(* CODESYS project CoreComponents.library
   Version: 1.3.1
   Title: CoreComponents
   DefaultNamespace: CoreComponents
   Placeholder: CoreComponents
   Company: Beckhoff Automation LLC

Project tree, tasks and I/O mapping:
  libraries: Tc2_DataExchange, * (Beckhoff Automation GmbH); Tc2_EtherCAT, * (Beckhoff Automation GmbH); Tc2_IoFunctions, * (Beckhoff Automation GmbH); Tc2_Math, * (Beckhoff Automation GmbH); Tc2_SerialCom, * (Beckhoff Automation GmbH); Tc2_Standard, * (Beckhoff Automation GmbH); Tc2_System, * (Beckhoff Automation GmbH); Tc2_TcpIp, * (Beckhoff Automation GmbH); Tc2_Utilities, * (Beckhoff Automation GmbH); Tc3_EventLogger, * (Beckhoff Automation GmbH); Tc3_JsonXml, * (Beckhoff Automation GmbH); Tc3_Module, * (Beckhoff Automation GmbH); Core, 1.3.0 (Beckhoff Automation LLC)
  Components/
    ADS/
      Interface/
        interface I_AdsAccess: AdsRW
        interface I_AdsRW: AmsNetId, AmsPort, Read, ReadBySymbol, Write, WriteBySymbol
      function block AdsReadWrite [ST]: Busy, Error, ErrorId, AdsComMode, AmsNetId, AmsPort, CyclicLogic, Read, ReadBySymbol, Write, WriteBySymbol
    Analog/
      DUT/
        data type ST_AnalogInputStatus_EL30xx
        data type ST_AnalogInputStatus_Generic
      Interface/
        interface I_AnalogChannel_Generic: DataValid, Error, Overrange, Underrange
        interface I_AnalogChannel_Standard: Limit1High, Limit1Low, Limit2High, Limit2Low
        interface I_AnalogInput: RawValue, Value
        interface I_AnalogOutput: RawValue, Value
      function block AnalogInput [ST]: CalibrateCustom, CalibrateLinear, FB_Init, Force, ForceValue, RawValue, Scale, Value
      function block AnalogInput_Generic [ST]: DataValid, Error, FB_Init, Overrange, Underrange
      function block AnalogInput_Standard [ST]: DataValid, Error, FB_Init, Limit1High, Limit1Low, Limit2High, Limit2Low, Overrange, Underrange
      function block AnalogOutput [ST]: CalibrateCustom, CalibrateLinear, FB_Init, Force, ForceValue, RawValue, Scale, Value
    CoE/
      DUT/
        data type ST_TerminalProductInfo
      Interface/
        interface I_CoeAccess: CoE
        interface I_CoeDevice: AdsAddr, Read, Write
      function block CoeDevice [ST]: Busy, Error, ErrorId, AdsAddr, CyclicLogic, Read, Write
      function block NullCoeDevice [ST]: AdsAddr, Busy, CyclicLogic, Error, ErrorId, Read, Write
    Cylinder/
      DUT/
        data type E_CylinderErrorId
        data type E_CylinderState
        data type ST_Cylinder_HMI
      Interface/
        interface I_Cylinder: ExtendTimeout, RetractTimeout
        interface I_CylinderCommand: Extend, Retract
        interface I_CylinderStatus: Extended, Extending, Retracted, Retracting
      function block Cylinder [ST]: CyclicLogic, Busy, Error, ErrorId, Extend, Extended, Extending, ExtendTimeout, Retract, Retracted, Retracting, RetractTimeout, Reset, FB_Init
      function block Cylinder_HMI [ST]: ExtendPermissive, RetractPermissive, ControlObject, CyclicLogic, ExtendCommandName, ExtendedName, FB_Init, RetractCommandName, RetractedName
      function block Cylinder_TcEvents [ST]: GetHighestActiveEventReaction, GetHighestActiveEventSeverity, Reset, SetEventReactions, CyclicLogic, FB_Init
    Digital/
      DUT/
        data type ST_DigitalInput_HMI
        data type ST_DigitalOutput_HMI
      Interface/
        interface I_DigitalInput: IsActive
        interface I_DigitalOutput: On
      Visitor/
        function block ForceVisitor [ST]: Force, VisitComponent
        function block ReleaseAllForceVisitor [ST]: ReleaseForces, VisitComponent, VisitModule
      function block DigitalInput_Combiner [ST]: AddInput, Force, IsActive
      function block DigitalInput_DebounceFallingEdge [ST]: CyclicLogic, DebounceTime, FB_Init, Force, IsActive
      function block DigitalInput_DebounceRisingEdge [ST]: CyclicLogic, DebounceTime, FB_Init, Force, IsActive
      function block DigitalInput_HMI [ST]: ControlObject, CyclicLogic, FB_Init
      function block DigitalInput_NC [ST]: FB_Init, Force, IsActive
      function block DigitalInput_NO [ST]: FB_Init, Force, IsActive
      function block DigitalOutput [ST]: FB_Init, Force, On
      function block DigitalOutput_HMI [ST]: ControlObject, CyclicLogic, FB_Init
    EtherCat/
      DUT/
        global variables EtherCatParameter
        data type ST_EtherCatMasterInfo
        data type ST_EtherCatSyncUnitTaskInfo
      Interface/
        interface I_EcIoDevice: Bootstrap, Configuration, DeviceError, Disabled, Init, InitCmdError, InvalidVPRS, OP, PreOp, SafeOp, State
        interface I_EtherCatDiagnosticEventProvider: RaiseEtherCatDiagnosticEvent, RaiseSyncUnitEvent
        interface I_EtherCatMasterDiagnostic: ConfiguredSlaveCount, GetIoDeviceByAddr, GetIoDeviceByName, LocalAmsNetId, MasterAmsNetId, RegisterEventProvider, SlaveCount
        interface I_IoDevice: IoDataValid
        interface I_SyncUnitTask: IoDataValid, IsHotConnect, SlaveCount
      function block EtherCatIoDevice [ST]: Bootstrap, CoE, Configuration, DeviceError, Disabled, Init, InitCmdError, InvalidVPRS, IoDataValid, OP, PreOp, SafeOp, State, AmsNetId, CyclicLogic, SyncUnit
      function block EtherCatMaster [ST]: FramesWcStatesOk, LookupMasterState, LookupSlaveState, MasterState, SlaveState, ConfiguredSlaveCount, GetIoDeviceByAddr, GetIoDeviceByName, LocalAmsNetId, MasterAmsNetId, RegisterEventProvider, SlaveCount, Initialize, Initialized, Reset, Busy, Error, ErrorId, CyclicLogic, FB_Init, Simulated
      function block EtherCatMaster_TcEvents [ST]: GetHighestActiveEventReaction, GetHighestActiveEventSeverity, RaiseEtherCatDiagnosticEvent, RaiseSyncUnitEvent, Reset, SetEventReactions, FB_Init
      function block SyncUnitTask [ST]: Initialize, Initialized, IoDataValid, IsHotConnect, IsTerminalPartOfSyncUnit, SlaveCount, Busy, Error, ErrorId, CyclicLogic, EventProvider, FB_Init, Simulated
    Recipe/
      Interface/
        interface I_RecipeManagment: AutoLoadChangesToActive, ChangesPending, LoadChangesToActive
      function block RecipeManagment [ST]: CyclicLogic, CompareData, AutoLoadChangesToActive, ChangesPending, LoadChangesToActive, FB_Init
    Safety/
      DUT/
        data type E_SafetyConnection_State
        data type E_SafetyEdm_State
        data type E_SafetyEStop_State
        data type E_SafetyGroup_Diag
        data type E_SafetyGroup_State
        data type E_SafetyMon_State
        data type E_SafetyOrAnd_State
        data type ST_SafetyAddressInfo
        data type ST_SafetyDeviceInfo
        data type ST_SafetyStateDiag
      Interface/
        interface I_InSafetyGroup: SafetyGroup
        interface I_SafetyBase: OK, ResetFunction
        interface I_SafetyModule: AddSafetyComponent, OK, SafetyPlcCoE
        interface I_SafetyReset: Execute, PulseDuration
        interface I_SafetySimulation: SimulateSafetyDiag, SimulateSafetyState
      Reset Function/
        function block SafetyResetPulse [ST]: CyclicLogic, Busy, Error, ErrorId, Execute, PulseDuration
      Visitor/
        function block SafetyOkVisitor [ST]: Check, OK, VisitComponent
        function block SetSafetySimulationVisitor [ST]: Diag, Simulated, State, VisitComponent
      function block SafetyAndOrFB [ST]: CyclicLogic
      function block SafetyBase [ST]: CyclicLogic, OK, Reset, ResetFunction, Simulated, SimulateSafetyDiag, SimulateSafetyState, Busy, Error, ErrorId
      function block SafetyConnectionFB_TcEvents [ST]: CyclicLogic, GetHighestActiveEventReaction, GetHighestActiveEventSeverity, Reset, SetEventReactions, FB_Init
      function block SafetyEdmFB_TcEvents [ST]: CyclicLogic, GetHighestActiveEventReaction, GetHighestActiveEventSeverity, Reset, SetEventReactions, FB_Init, SafetyGroup
      function block SafetyEstopFB_TcEvents [ST]: CyclicLogic, GetHighestActiveEventReaction, GetHighestActiveEventSeverity, Reset, SetEventReactions, ActiveName, FB_Init, SafetyGroup
      function block SafetyGroup_TcEvents [ST]: CyclicLogic, GetHighestActiveEventReaction, GetHighestActiveEventSeverity, Reset, SetEventReactions, AutoResetFaults, FB_Init
      function block SafetyModule [ST]: OnCyclicCall, Initializing, Simulated, SimulateSafetyDiag, SimulateSafetyState, Busy, Error, ErrorId, AddSafetyComponent, FB_Init, OK, Reset, SafetyAddressInfo, SafetyPlcCoE
      function block SafetyMonFB_TcEvents [ST]: CyclicLogic, GetHighestActiveEventReaction, GetHighestActiveEventSeverity, Reset, SetEventReactions, ActiveAlarm, ActiveName, FB_Init, SafetyGroup
    Serial/
      Interface/
        interface I_SerialByteConnection: ByteData, ByteDataRecieved, SendAByte
        interface I_SerialLineControl: rxBuffer, txBuffer
        interface I_SerialStringConnection: SendAString, StringData, StringRecieved
      function block SerialByteConnection [ST]: ByteData, ByteDataRecieved, CyclicLogic, FB_Init, Reset, SendAByte, SetDependencies
      function block SerialLineControl_ADS [ST]: CyclicLogic, rxBuffer, SetConnectionConfig, txBuffer
      function block SerialLineControl_Terminal [ST]: CyclicLogic, FB_Init, rxBuffer, SetConnectionConfig, SetDependencies, txBuffer
      function block SerialStringConnection [ST]: CyclicLogic, FB_Init, Reset, SendAString, SetDependencies, SetSerialConfiguration, StringData, StringRecieved
    Tcp Ip/
      DUT/
        data type ST_TcpIpPayload
      Interface/
        interface I_TcpIpConnection: ConnectionState, IP, Port, RegisterCommand, SendCommand, SendPriorityCommand, Socket
        interface I_TcpIpSubscription: UpdateCommandResult
      function block TcpIpCommandResultFilter [ST]: CyclicLogic, FB_Init, UpdateCommandResult
      function block TcpIpConnection [ST]: CyclicLogic, Initialize, Initialized, EvaluateResponse, GetNextCommand, GetNextPriorityCommand, SendReceiveSequence, ConnectionState, IP, PollTime, Port, ReceiveTimeout, ReconnectionTime, RegisterCommand, SendCommand, SendInterval, SendPriorityCommand, Socket
      global variables TcpIpConnectionParameter
  Project Information/
    function F_GetCompany [ST]
    function F_GetTitle [ST]
    function F_GetVersion [ST]
  Utilities/
    AnyBuffer/
      DUT/
        data type ST_BufferConfiguration
        data type ST_BufferMetadata
      Interface/
        interface I_AnyBuffer: Clear, Configuration, DeleteAtIndex, isEmpty, isFull, Metadata, PeekAtIndex, PopAtIndex, PopLeft, PopRight, PushAtIndex, PushLeft, PushRight, ReplaceAtIndex
        interface I_AnyBufferStrategy: Clear, isEmpty, isFull
      TypedBuffers/
        function block FifoBuffer [ST]: Clear, FB_Init, isEmpty, isFull, Pop, Push
        function block LifoBuffer [ST]: Clear, FB_Init, isEmpty, isFull, Pop, Push
        function block ListBuffer [ST]: Clear, FB_Init, isEmpty, isFull, Pop, Push, removeOldest
        function block RingBuffer [ST]: AdvanceHead, AdvanceTail, Clear, FB_Init, isEmpty, isFull, Pop, Push
      function block AnyBuffer [ST]: buffer, Clear, Configuration, CountDecrement, CountIncrement, DeleteAtIndex, FB_Exit, FB_Init, FB_Reinit, isEmpty, isFull, Metadata, PeekAtIndex, PopAtIndex, PopLeft, PopRight, PushAtIndex, PushLeft, PushRight, ReplaceAtIndex
    File/
      DUT/
        data type ST_File_HMI
      Interface/
        interface I_FileHandler: ClearDocument, Datatype, LoadFile, nData, Path, pData, ReadSymbol, SaveFile, SymbolName, Timeout, UpdateSymbol
      function block File_HMI [ST]: LoadPermissive, SavePermissive, ControlObject, CyclicLogic, FB_Init
      function block JsonFile [ST]: CyclicLogic, ClearDocument, Datatype, LoadFile, nData, Path, pData, ReadSymbol, SaveFile, SymbolName, Timeout, UpdateSymbol, LoadFileSequence, SaveFileSequence, Reset, Busy, Error, ErrorId
      function block StringHelper [ST]: GetExtensionOrVarName, GetFileNameFromPath, GetFilePath, GetName, GetPath, GetSymbolPath, RemoveFirstChar, RemoveLastChar, StringToCharArray, ValidInput
    Flash/
      function block SyncedSquareWaves [ST]: Initialize, Initialized, CyclicLogic, Wave_0_5Hz, Wave_100Hz, Wave_1Hz, Wave_2Hz, Wave_500Hz, Wave_50Hz, Wave_5Hz
    Force/
      DUT/
        data type E_ForceState
      Interface/
        interface I_ForcibleBool: Force
        interface I_ForcibleInt: Force, ForceValue
      function block ForcibleBool [ST]: ResolveOutput, CurrentForceState, FB_Init, Input, Output, SetForceState
      function block ForcibleInt [ST]: ResolveOutput, CurrentForceState, FB_Init, ForceValue, Input, Output, SetForceState
    Functions/
      function CompareLREAL [ST]
      function CompareModulo [ST]
      function PercentToAnalog [ST]
    Scaling/
      Interface/
        interface I_AnalogScalable: Scale
        interface I_AnalogScale: InputMaximum, InputMinimum, OutputMaximum, OutputMinimum
        interface I_CalibratableLinear: CalibrateLinear
        interface I_CalibrateLinear: Gain, Offset
        interface I_TransformLRealValue: Transform
      function block AnalogScale [ST]: InputMaximum, InputMinimum, OutputMaximum, OutputMinimum, Transform
      function block Calibrate [ST]: Gain, Offset, Transform
    Timing/
      function block Stopwatch [ST]: Elapsed, Lap, Running, Start, Stop
  Version/
    global variables Global_Version
*)

// Components/Analog/DUT/ST_AnalogInputStatus_EL30xx
{attribute 'pack_mode' := '1'}
TYPE ST_AnalogInputStatus_EL30xx :
	STRUCT
		Underrrange : BIT;
		Overrange	: BIT;
		Limit1L		: BIT;
		Limit1H		: BIT;
		Limit2L		: BIT;
		Limit2H		: BIT;
		Error		: BIT;
		TxPDOState	: BIT;
		TxPDOToggle : BIT;
	END_STRUCT
END_TYPE

// Components/Analog/DUT/ST_AnalogInputStatus_Generic
{attribute 'pack_mode' := '1'}
TYPE ST_AnalogInputStatus_Generic :
	STRUCT
		Underrrange : BIT;
		Overrange	: BIT;
		Error		: BIT;
		WcState		: BIT;
	END_STRUCT
END_TYPE

// Components/CoE/DUT/ST_TerminalProductInfo
{attribute 'pack_mode' := '2'}
TYPE ST_TerminalProductInfo : // Parameter 16#1018:0
	STRUCT
		Identity	 : WORD;
		VendorId	 : DINT;
		ProductCode	 : DINT;
		Revision	 : DINT;
		SerialNumber : DINT;
	END_STRUCT
END_TYPE

// Components/Cylinder/DUT/E_CylinderErrorId
{attribute 'qualified_only'}
TYPE E_CylinderErrorId : (
		NoError				  := 0,
		ExtendTimeout		  := 1,
		RetractTimeout		  := 2,
		ExtendedPlausibility  := 3,
		RetractedPlausibility := 4,
		BothSensorsActive	  := 5
	) UDINT;
END_TYPE

// Components/Cylinder/DUT/E_CylinderState
{attribute 'qualified_only'}
TYPE E_CylinderState : (
		Undefined  := 0,
		Extending  := 1,
		Extended   := 2,
		Retracting := 3,
		Retracted  := 4
	);
END_TYPE

// Components/Cylinder/DUT/ST_Cylinder_HMI
TYPE ST_Cylinder_HMI EXTENDS ST_HmiFunction :
	STRUCT
		Busy		  : BOOL;
		Error		  : BOOL;
		ErrorId		  : UDINT;
		Extended	  : BOOL;
		ExtendedName  : STRING := 'Extended';
		Retracted	  : BOOL;
		RetractedName : STRING := 'Retracted';
		Extend		  : Button;
		Retract		  : Button;
	END_STRUCT
END_TYPE

// Components/Digital/DUT/ST_DigitalInput_HMI
TYPE ST_DigitalInput_HMI EXTENDS ST_HmiFunction :
	STRUCT
		Active : BOOL;
		Force  : E_ForceState;
	END_STRUCT
END_TYPE

// Components/Digital/DUT/ST_DigitalOutput_HMI
TYPE ST_DigitalOutput_HMI EXTENDS ST_HmiFunction :
	STRUCT
		On	  : BOOL;
		Force : E_ForceState;
	END_STRUCT
END_TYPE

// Components/EtherCat/DUT/ST_EtherCatMasterInfo
TYPE ST_EtherCatMasterInfo :
	STRUCT
		AmsNetID	  : AMSNETID;
		DevID		  : UINT;
		DevState	  : UINT;
		ChangeCount	  : UINT;
		SlaveCount	  : UINT;
		CfgSlaveCount : UINT;
	END_STRUCT
END_TYPE

// Components/EtherCat/DUT/ST_EtherCatSyncUnitTaskInfo
TYPE ST_EtherCatSyncUnitTaskInfo :
	STRUCT
		WcState	   : BIT;
		ObjectId   : OTCID;
		State	   : UINT;
		SlaveCount : UINT;
	END_STRUCT
END_TYPE

// Components/Safety/DUT/E_SafetyConnection_State
{attribute 'qualified_only'}
{attribute 'strict'}
TYPE E_SafetyConnection_State : (
		Reset	   := 100,
		Session	   := 101,
		Connection := 102,
		Parameter  := 103,
		Data	   := 104,
		Shutdown   := 105,
		Deactive   := 106
	) USINT;
END_TYPE

// Components/Safety/DUT/E_SafetyEdm_State
{attribute 'qualified_only'}
TYPE E_SafetyEdm_State : (
		Invalid := 0,
		Stop	:= 2,
		Error	:= 4,
		Reset	:= 5,
		MonOff	:= 14,
		MonOn	:= 15
	) USINT;
END_TYPE

// Components/Safety/DUT/E_SafetyEStop_State
{attribute 'qualified_only'}
TYPE E_SafetyEStop_State : (
		Invalid	 := 0,
		Run		 := 1,
		Stop	 := 2,
		Safe	 := 3,
		Error	 := 4,
		Reset	 := 5,
		Start	 := 6,
		DelayOut := 7
	) USINT;
END_TYPE

// Components/Safety/DUT/E_SafetyGroup_Diag
{attribute 'qualified_only'}
TYPE E_SafetyGroup_Diag : (
		NoError		  := 0,
		FbError		  := 1,
		ComError	  := 2,
		ModuleError	  := 3,
		CmpError	  := 4,
		DeactiveError := 5,
		RestartError  := 6
	) UINT;
END_TYPE

// Components/Safety/DUT/E_SafetyGroup_State
{attribute 'qualified_only'}
TYPE E_SafetyGroup_State : (
		Invalid		 := 0,
		Run			 := 1,
		Stop		 := 2,
		Error		 := 4,
		Reset		 := 5,
		Start		 := 6,
		StopError	 := 7,
		Deactive	 := 16,
		WaitComError := 17
	) USINT;
END_TYPE

// Components/Safety/DUT/E_SafetyMon_State
{attribute 'qualified_only'}
TYPE E_SafetyMon_State : (
		Invalid	   := 0,
		Run		   := 1,
		Stop	   := 2,
		Safe	   := 3,
		Error	   := 4,
		Reset	   := 5,
		Start	   := 6,
		ErrorDelay := 7,
		DelayOut   := 8,
		FuncTest   := 9
	) USINT;
END_TYPE

// Components/Safety/DUT/E_SafetyOrAnd_State
{attribute 'qualified_only'}
TYPE E_SafetyOrAnd_State : (
		Invalid := 0,
		Run		:= 1,
		Stop	:= 2,
		Safe	:= 3
	) USINT;
END_TYPE

// Components/Safety/DUT/ST_SafetyAddressInfo
{attribute 'pack_mode' := '2'}
TYPE ST_SafetyAddressInfo : // Parameter 16#F980:0
	STRUCT
		FSoEAddress		  : WORD;
		SerialNumber	  : DINT;
		ProjectCRC		  : WORD;
		DefaultProjectCRC : WORD;
	END_STRUCT
END_TYPE

// Components/Safety/DUT/ST_SafetyDeviceInfo
{attribute 'pack_mode' := '2'}
TYPE ST_SafetyDeviceInfo : // Parameter 16#F9C0:0
	STRUCT
		DeviceName			 : STRING;
		SoftwareVersion		 : STRING;
		BootloaderVersion	 : STRING;
		SoftwareChecksum	 : DINT;
		BootmanagerChecksum	 : DINT;
		BootloaderChecksum	 : DINT;
		TwinSAFELogicVersion : DINT;
	END_STRUCT
END_TYPE

// Components/Safety/DUT/ST_SafetyStateDiag
{attribute 'pack_mode' := '1'}
TYPE ST_SafetyStateDiag :
	STRUCT
		State : USINT;
		Diag  : UINT; // **NOT PRESENT ON AND/OR FBs ** For components with USINT as Diag connection, connect first 8 Bit of UINT Diag. Inherited FB is evaluating correct length.
	END_STRUCT
END_TYPE

// Components/Tcp Ip/DUT/ST_TcpIpPayload
TYPE ST_TcpIpPayload :
	STRUCT
		Size : UDINT;
		Data : ARRAY[0..(TcpIpConnectionParameter.PayloadSize - 1)] OF BYTE;
	END_STRUCT
END_TYPE

// Utilities/AnyBuffer/DUT/ST_BufferConfiguration
TYPE ST_BufferConfiguration :
	STRUCT
		isPersistent	 : BOOL; // is the buffer persistent?
		capacity		 : DINT; // No of elements in buffer
		elementSize		 : DINT; // Buffer element size in bytes
		bufferSize		 : DINT; // Complete buffer size in bytes	
		bufferBoundLower : DINT; // Lower boundary of the buffer
		bufferBoundUpper : DINT; // Upper boundary of the buffer	
	END_STRUCT
END_TYPE

// Utilities/AnyBuffer/DUT/ST_BufferMetadata
TYPE ST_BufferMetadata :
	STRUCT
		headIndex	 : DINT;
		tailIndex	 : DINT;
		capacity	 : DINT;
		elementCount : DINT;
	END_STRUCT
END_TYPE

// Utilities/File/DUT/ST_File_HMI
TYPE ST_File_HMI EXTENDS ST_HmiFunction :
	STRUCT
		Path	: STRING;
		Load	: Button;
		Save	: Button;
		NewPath : BOOL;
	END_STRUCT
END_TYPE

// Utilities/Force/DUT/E_ForceState
{attribute 'qualified_only'}
{attribute 'strict'}
{attribute 'to_string'}
TYPE E_ForceState : (
		Unforced := 0,
		ForceOn	 := 1,
		ForceOff := 2
	) DINT;
END_TYPE

// Components/EtherCat/DUT/EtherCatParameter
VAR_GLOBAL CONSTANT
	MAX_EC_SLAVES : UINT := 49;
END_VAR

// Components/Tcp Ip/TcpIpConnectionParameter
{attribute 'qualified_only'}
VAR_GLOBAL CONSTANT
	PayloadSize : UDINT := 1460; // Payload in Bytes
END_VAR

// Version/Global_Version
{attribute 'TcGenerated'}
{attribute 'no-analysis'}
{attribute 'linkalways'}
// This function has been automatically generated from the project information.
VAR_GLOBAL CONSTANT
	{attribute 'const_non_replaced'}
	stLibVersion_CoreComponents : ST_LibVersion := (iMajor := 1, iMinor := 3, iBuild := 1, iRevision := 0, nFlags := 0, sVersion := '1.3.1');
END_VAR

// Components/ADS/Interface/I_AdsAccess
INTERFACE I_AdsAccess EXTENDS I_Base

PROPERTY AdsRW : I_AdsRW
GET
END_GET
SET
END_SET
END_PROPERTY

END_INTERFACE

// Components/ADS/Interface/I_AdsRW
INTERFACE I_AdsRW EXTENDS I_Component, I_TaskResult

{attribute 'monitoring' := 'call'}
PROPERTY AmsNetId : T_AmsNetId
GET
END_GET
SET
END_SET
END_PROPERTY

{attribute 'monitoring' := 'call'}
PROPERTY AmsPort : T_AmsPort
GET
END_GET
SET
END_SET
END_PROPERTY

METHOD Read
VAR_INPUT
	IdxGrp	  : UDINT;
	IdxOffset : UDINT;
	pDestAddr : PVOID;
	Length	  : UDINT;
END_VAR
END_METHOD

METHOD ReadBySymbol
VAR_INPUT
	SymbolName : STRING(255);
	pDestAddr  : PVOID;
	Length	   : UDINT;
END_VAR
END_METHOD

METHOD Write
VAR_INPUT
	IdxGrp		: UDINT;
	IdxOffset	: UDINT;
	pSourceAddr : PVOID;
	Length		: UDINT;
END_VAR
END_METHOD

METHOD WriteBySymbol
VAR_INPUT
	SymbolName	: STRING(255);
	pSourceAddr : PVOID;
	Length		: UDINT;
END_VAR
END_METHOD

END_INTERFACE

// Components/ADS/AdsReadWrite
FUNCTION_BLOCK AdsReadWrite EXTENDS CyclicComponent IMPLEMENTS I_AdsRW
VAR
	{attribute 'hide'}
	_AmsNetId : T_AmsNetId;
	{attribute 'hide'}
	_AmsPort : T_AmsPort;
	{attribute 'hide'}
	_AdsComMode		  : E_AdsComMode := eAdsComModeSecureCom;
	AdsRead			  : ADSREAD;
	AdsWrite		  : ADSWRITE;
	ReadAdsSymByName  : FB_ReadAdsSymByName;
	WriteAdsSymByName : FB_WriteAdsSymByName;
END_VAR

{attribute 'monitoring' := 'call'}
PROPERTY Busy : BOOL
GET
Busy := AdsWrite.BUSY OR AdsRead.BUSY OR ReadAdsSymByName.bBusy OR WriteAdsSymByName.bBusy;
END_GET
END_PROPERTY

{attribute 'monitoring' := 'call'}
PROPERTY Error : BOOL
GET
Error := AdsWrite.ERR OR AdsRead.ERR OR ReadAdsSymByName.bError OR WriteAdsSymByName.bError;
END_GET
END_PROPERTY

{attribute 'monitoring' := 'call'}
PROPERTY ErrorId : UDINT
GET
IF AdsWrite.ERR THEN
	ErrorID := AdsWrite.ERRID;
ELSIF AdsRead.ERR THEN
	ErrorID := AdsRead.ERRID;
ELSIF ReadAdsSymByName.bError THEN
	ErrorID := ReadAdsSymByName.nErrorId;
ELSIF WriteAdsSymByName.bError THEN
	ErrorID := WriteAdsSymByName.nErrorId;
ELSE
	ErrorID := 0;
END_IF
END_GET
END_PROPERTY

PROPERTY AdsComMode : E_AdsComMode
SET
_AdsComMode := AdsComMode;
END_SET
END_PROPERTY

{attribute 'monitoring' := 'call'}
PROPERTY AmsNetId : T_AmsNetId
GET
AmsNetId := _AmsNetId;
END_GET
SET
_AmsNetId := AmsNetId;
END_SET
END_PROPERTY

{attribute 'monitoring' := 'call'}
PROPERTY AmsPort : T_AmsPort
GET
AmsPort := _AmsPort;
END_GET
SET
_AmsPort := AmsPort;
END_SET
END_PROPERTY

METHOD CyclicLogic
AdsRead(NETID := _AmsNetId, PORT := _AmsPort, TMOUT := DEFAULT_ADS_TIMEOUT);
AdsRead.READ := FALSE;
AdsWrite(NETID := _AmsNetId, PORT := _AmsPort, TMOUT := DEFAULT_ADS_TIMEOUT);
AdsWrite.WRITE := FALSE;

//
ReadAdsSymByName(sNetId		   := _AmsNetId,
				 nPort		   := _AmsPort,
				 tTimeout	   := DEFAULT_ADS_TIMEOUT,
				 eComMode	   := _AdsComMode,
				 bClearOnError := TRUE);

ReadAdsSymByName.bRead := FALSE;

//
WriteAdsSymByName(sNetId   := _AmsNetId,
				  nPort	   := _AmsPort,
				  tTimeout := DEFAULT_ADS_TIMEOUT,
				  eComMode := _AdsComMode);

WriteAdsSymByName.bWrite := FALSE;
END_METHOD

METHOD Read
VAR_INPUT
	IdxGrp	  : UDINT;
	IdxOffset : UDINT;
	pDestAddr : PVOID;
	Length	  : UDINT;
END_VAR
IF AdsRead.BUSY THEN
	RETURN;
END_IF

AdsRead.IDXGRP	 := IdxGrp;
AdsRead.IDXOFFS	 := IdxOffset;
AdsRead.LEN		 := Length;
AdsRead.DESTADDR := pDestAddr;
AdsRead.READ	 := TRUE;
END_METHOD

METHOD ReadBySymbol
VAR_INPUT
	SymbolName : STRING(255);
	pDestAddr  : PVOID;
	Length	   : UDINT;
END_VAR
IF ReadAdsSymByName.bBusy THEN
	RETURN;
END_IF

ReadAdsSymByName.sVarName  := SymbolName;
ReadAdsSymByName.nDestAddr := pDestAddr;
ReadAdsSymByName.nLen	   := Length;
ReadAdsSymByName.bRead	   := TRUE;
END_METHOD

METHOD Write
VAR_INPUT
	IdxGrp		: UDINT;
	IdxOffset	: UDINT;
	pSourceAddr : PVOID;
	Length		: UDINT;
END_VAR
IF AdsWrite.BUSY THEN
	RETURN;
END_IF

AdsWrite.IDXGRP	 := IdxGrp;
AdsWrite.IDXOFFS := IdxOffset;
AdsWrite.LEN	 := Length;
AdsWrite.SRCADDR := pSourceAddr;
AdsWrite.WRITE	 := TRUE;
END_METHOD

METHOD WriteBySymbol
VAR_INPUT
	SymbolName	: STRING(255);
	pSourceAddr : PVOID;
	Length		: UDINT;
END_VAR
IF WriteAdsSymByName.bBusy THEN
	RETURN;
END_IF

WriteAdsSymByName.sVarName := SymbolName;
WriteAdsSymByName.nSrcAddr := pSourceAddr;
WriteAdsSymByName.nLen	   := Length;
WriteAdsSymByName.bWrite   := TRUE;
END_METHOD

END_FUNCTION_BLOCK

// Components/Analog/Interface/I_AnalogChannel_Generic
INTERFACE I_AnalogChannel_Generic EXTENDS I_AnalogInput

PROPERTY DataValid : BOOL
GET
END_GET
END_PROPERTY

PROPERTY Error : BOOL
GET
END_GET
END_PROPERTY

PROPERTY Overrange : BOOL
GET
END_GET
END_PROPERTY

PROPERTY Underrange : BOOL
GET
END_GET
END_PROPERTY

END_INTERFACE

// Components/Analog/Interface/I_AnalogInput
INTERFACE I_AnalogInput EXTENDS I_Component, I_ForcibleInt

{attribute 'monitoring' := 'call'}
PROPERTY RawValue : INT
GET
END_GET
END_PROPERTY

{attribute 'monitoring' := 'call'}
PROPERTY Value : LREAL
GET
END_GET
END_PROPERTY

END_INTERFACE

// Utilities/Force/Interface/I_ForcibleInt
INTERFACE I_ForcibleInt

{attribute 'monitoring' := 'call'}
PROPERTY Force : E_ForceState
GET
END_GET
SET
END_SET
END_PROPERTY

PROPERTY ForceValue : INT
GET
END_GET
SET
END_SET
END_PROPERTY

END_INTERFACE

// Components/Analog/Interface/I_AnalogChannel_Standard
INTERFACE I_AnalogChannel_Standard EXTENDS I_AnalogChannel_Generic

PROPERTY Limit1High : BOOL
GET
END_GET
END_PROPERTY

PROPERTY Limit1Low : BOOL
GET
END_GET
END_PROPERTY

PROPERTY Limit2High : BOOL
GET
END_GET
END_PROPERTY

PROPERTY Limit2Low : BOOL
GET
END_GET
END_PROPERTY

END_INTERFACE

// Components/Analog/Interface/I_AnalogOutput
INTERFACE I_AnalogOutput EXTENDS I_Component, I_ForcibleInt

{attribute 'monitoring' := 'call'}
PROPERTY RawValue : INT
GET
END_GET
SET
END_SET
END_PROPERTY

{attribute 'monitoring' := 'call'}
PROPERTY Value : LREAL
GET
END_GET
SET
END_SET
END_PROPERTY

END_INTERFACE

// Components/Analog/AnalogInput
FUNCTION_BLOCK AnalogInput EXTENDS Component IMPLEMENTS I_AnalogInput, I_AnalogScalable, I_CalibratableLinear
VAR
	Input			 : REFERENCE TO INT;
	Forcible		 : ForcibleInt(_Name);
	_Scale			 : I_AnalogScale;
	_CalibrateLinear : I_CalibrateLinear;
	_CalibrateCustom : I_TransformLRealValue;
END_VAR

VAR
	{attribute 'hide'}
	DefaultScale : AnalogScale;
	{attribute 'hide'}
	DefaultCalibration : Calibrate;
END_VAR

PROPERTY CalibrateCustom : I_TransformLrealValue
SET
_CalibrateCustom := CalibrateCustom;
END_SET
END_PROPERTY

PROPERTY CalibrateLinear : I_CalibrateLinear
GET
CalibrateLinear := _CalibrateLinear;
END_GET
SET
_CalibrateLinear := CalibrateLinear;
END_SET
END_PROPERTY

(*FB_Init is always available implicitly and it is used primarily for initialization.
The return value is not evaluated. For a specific influence, you can also declare the
methods explicitly and provide additional code there with the standard initialization
code. You can evaluate the return value.*)
METHOD FB_Init : BOOL
VAR_INPUT
	(* TRUE: the retain variables are initialized (reset warm / reset cold)*)
	bInitRetains : BOOL;

	(* TRUE: the instance will be copied to the copy code afterward (online change)   *)
	bInCopyCode : BOOL;
	Name		: Core.T_MaxString;
	Input		: REFERENCE TO INT;
END_VAR
_Scale			 := DefaultScale;
_CalibrateLinear := DefaultCalibration;
THIS^.Input		 REF= Input;
END_METHOD

{attribute 'monitoring' := 'call'}
PROPERTY Force : E_ForceState
GET
Force := Forcible.CurrentForceState;
END_GET
SET
VAR
	ForceString : T_MaxString := TO_STRING(Force);
END_VAR
Forcible.SetForceState(Force);
END_SET
END_PROPERTY

PROPERTY ForceValue : INT
GET
ForceValue := Forcible.ForceValue;
END_GET
SET
Forcible.ForceValue := ForceValue;
END_SET
END_PROPERTY

{attribute 'monitoring' := 'call'}
PROPERTY RawValue : INT
GET
Forcible.Input := Input;
RawValue	   := Forcible.Output;
END_GET
END_PROPERTY

PROPERTY Scale : I_AnalogScale
GET
Scale := _Scale;
END_GET
SET
_Scale := Scale;
END_SET
END_PROPERTY

{attribute 'monitoring' := 'call'}
PROPERTY Value : LREAL
GET
IF _CalibrateCustom = 0 THEN
	Value := _CalibrateLinear.Transform(_Scale.Transform(RawValue));
ELSE
	Value := _CalibrateCustom.Transform(_Scale.Transform(RawValue));
END_IF
END_GET
END_PROPERTY

END_FUNCTION_BLOCK

// Utilities/Scaling/Interface/I_AnalogScalable
INTERFACE I_AnalogScalable EXTENDS I_Base

PROPERTY Scale : I_AnalogScale
GET
END_GET
SET
END_SET
END_PROPERTY

END_INTERFACE

// Utilities/Scaling/Interface/I_AnalogScale
INTERFACE I_AnalogScale EXTENDS I_TransformLrealValue

PROPERTY InputMaximum : LREAL
GET
END_GET
SET
END_SET
END_PROPERTY

PROPERTY InputMinimum : LREAL
GET
END_GET
SET
END_SET
END_PROPERTY

PROPERTY OutputMaximum : LREAL
GET
END_GET
SET
END_SET
END_PROPERTY

PROPERTY OutputMinimum : LREAL
GET
END_GET
SET
END_SET
END_PROPERTY

END_INTERFACE

// Utilities/Scaling/Interface/I_TransformLRealValue
INTERFACE I_TransformLRealValue EXTENDS I_Base

METHOD Transform : LREAL
VAR_INPUT
	Value	: LREAL;
	Reverse : BOOL := FALSE;
END_VAR
END_METHOD

END_INTERFACE

// Utilities/Scaling/Interface/I_CalibratableLinear
INTERFACE I_CalibratableLinear EXTENDS I_Base

PROPERTY CalibrateLinear : I_CalibrateLinear
GET
END_GET
SET
END_SET
END_PROPERTY

END_INTERFACE

// Utilities/Scaling/Interface/I_CalibrateLinear
INTERFACE I_CalibrateLinear EXTENDS I_TransformLrealValue

PROPERTY Gain : LREAL
SET
END_SET
END_PROPERTY

PROPERTY Offset : LREAL
SET
END_SET
END_PROPERTY

END_INTERFACE

// Utilities/Force/ForcibleInt
FUNCTION_BLOCK ForcibleInt
VAR
	Name			   : T_MaxString;
	_CurrentForceState : E_ForceState;
	ForceEvent		   : FB_TcAlarm;
	RequestedValue	   : INT;
	_Output			   : INT;
	_ForceValue : INT;
END_VAR

METHOD PRIVATE ResolveOutput
VAR
	ForceString : T_MaxString := TO_STRING(_CurrentForceState);
END_VAR
CASE _CurrentForceState OF
	E_ForceState.Unforced:
		_Output := RequestedValue;
		ForceEvent.Clear();

	E_ForceState.ForceOn:
		IF NOT ForceEvent.bActive THEN
			ForceEvent.ipArguments.Clear().AddString(Name).AddString(ForceString);
			ForceEvent.Raise();
		END_IF

		_Output := _ForceValue;

	E_ForceState.ForceOff:
		IF NOT ForceEvent.bActive THEN
			ForceEvent.ipArguments.Clear().AddString(Name).AddString(ForceString);
			ForceEvent.Raise();
		END_IF

		_Output := 0;
END_CASE
END_METHOD

{attribute 'monitoring' := 'call'}
PROPERTY CurrentForceState : E_ForceState
GET
CurrentForceState := _CurrentForceState;
END_GET
END_PROPERTY

//FB_Init is always available implicitly and it is used primarily for initialization.

//The return value is not evaluated. For a specific influence, you can also declare the

//methods explicitly and provide additional code there with the standard initialization

//code. You can evaluate the return value.
METHOD FB_Init : BOOL
VAR_INPUT
	bInitRetains : BOOL; // TRUE: the retain variables are initialized (reset warm / reset cold)
	bInCopyCode	 : BOOL; // TRUE: the instance will be copied to the copy code afterward (online change) 
	Name		 : T_MaxString;
END_VAR
THIS^.Name := Name;
{analysis -15}
IF NOT ForceEvent.EqualsToEventEntryEx(TC_EVENTS.IO.ForceActive) THEN
	ForceEvent.CreateEx(TC_EVENTS.IO.ForceActive, 0);
END_IF
END_METHOD

PROPERTY ForceValue : INT
GET
ForceValue := _ForceValue;
END_GET
SET
_ForceValue := ForceValue;
END_SET
END_PROPERTY

{attribute 'monitoring' := 'call'}
PROPERTY Input : INT
SET
RequestedValue := Input;
ResolveOutput();
END_SET
END_PROPERTY

{attribute 'monitoring' := 'call'}
PROPERTY Output : INT
GET
Output := _Output;
END_GET
END_PROPERTY

METHOD SetForceState
VAR_INPUT
	ForceState : E_ForceState;
END_VAR
IF ForceState = _CurrentForceState THEN
	RETURN;
END_IF

_CurrentForceState := ForceState;
ResolveOutput();
END_METHOD

END_FUNCTION_BLOCK

// Utilities/Scaling/AnalogScale
FUNCTION_BLOCK AnalogScale IMPLEMENTS I_AnalogScale
VAR
	_InputMinimum  : LREAL := -32768;
	_InputMaximum  : LREAL := 32767;
	_OutputMinimum : LREAL := -32768;
	_OutputMaximum : LREAL := 32767;
END_VAR

PROPERTY InputMaximum : LREAL
GET
InputMaximum := _InputMaximum;
END_GET
SET
_InputMaximum := InputMaximum;
END_SET
END_PROPERTY

PROPERTY InputMinimum : LREAL
GET
InputMinimum := _InputMinimum;
END_GET
SET
_InputMinimum := InputMinimum;
END_SET
END_PROPERTY

PROPERTY OutputMaximum : LREAL
GET
OutputMaximum := _OutputMaximum;
END_GET
SET
_OutputMaximum := OutputMaximum;
END_SET
END_PROPERTY

PROPERTY OutputMinimum : LREAL
GET
OutputMinimum := _OutputMinimum;
END_GET
SET
_OutputMinimum := OutputMinimum;
END_SET
END_PROPERTY

METHOD Transform : LREAL
VAR_INPUT
	Value	: LREAL;
	Reverse : BOOL := FALSE;
END_VAR

VAR_INST
	Slope : LREAL;
END_VAR
//Scale is invalid
IF _InputMinimum >= _InputMaximum THEN
	Transform := 0;
	RETURN;
ELSIF _OutputMinimum >= _OutputMaximum THEN
	Transform := 0;
	RETURN;
END_IF

//Input is invalid
IF Value <= _InputMinimum THEN
	Transform := _OutputMinimum;
	RETURN;
ELSIF Value >= _InputMaximum THEN
	Transform := _OutputMaximum;
	RETURN;
END_IF

//I/O ok--scale it
IF (_InputMaximum - _InputMinimum) <> 0.0 THEN
	Slope := (_OutputMaximum - _OutputMinimum) / (_InputMaximum - _InputMinimum);
ELSE
	Slope := 0.0;
END_IF

Transform := Slope * (Value - _InputMinimum) + _OutputMinimum;
END_METHOD

END_FUNCTION_BLOCK

// Utilities/Scaling/Calibrate
FUNCTION_BLOCK Calibrate IMPLEMENTS I_CalibrateLinear
VAR
	_Gain	: LREAL := 1;
	_Offset : LREAL := 0;
END_VAR

PROPERTY Gain : LREAL
SET
_Gain := Gain;
END_SET
END_PROPERTY

PROPERTY Offset : LREAL
SET
_Offset := Offset;
END_SET
END_PROPERTY

METHOD Transform : LREAL
VAR_INPUT
	Value	: LREAL;
	Reverse : BOOL := FALSE;
END_VAR
IF Reverse THEN
	Transform := (Value - _Offset) / _Gain;
ELSE
	Transform := Value * _Gain + _Offset;
END_IF
END_METHOD

END_FUNCTION_BLOCK

// Components/Analog/AnalogInput_Generic
FUNCTION_BLOCK AnalogInput_Generic EXTENDS AnalogInput IMPLEMENTS I_AnalogChannel_Generic
VAR
	Status : REFERENCE TO ST_AnalogInputStatus_Generic;
END_VAR

PROPERTY DataValid : BOOL
GET
DataValid := NOT Status.WcState;
END_GET
END_PROPERTY

PROPERTY Error : BOOL
GET
Error := Status.Error;
END_GET
END_PROPERTY

(*FB_Init is always available implicitly and it is used primarily for initialization.
The return value is not evaluated. For a specific influence, you can also declare the
methods explicitly and provide additional code there with the standard initialization
code. You can evaluate the return value.*)
METHOD FB_Init : BOOL
VAR_INPUT
	(* TRUE: the retain variables are initialized (reset warm / reset cold)*)
	bInitRetains : BOOL;

	(* TRUE: the instance will be copied to the copy code afterward (online change)   *)
	bInCopyCode : BOOL;
	Name		: T_MaxString;
	Input		: REFERENCE TO INT;
	Status		: REFERENCE TO ST_AnalogInputStatus_Generic;
END_VAR
THIS^.Status REF= Status;
END_METHOD

PROPERTY Overrange : BOOL
GET
Overrange := Status.Overrange;
END_GET
END_PROPERTY

PROPERTY Underrange : BOOL
GET
Underrange := Status.Underrrange;
END_GET
END_PROPERTY

END_FUNCTION_BLOCK

// Components/Analog/AnalogInput_Standard
FUNCTION_BLOCK AnalogInput_Standard EXTENDS AnalogInput IMPLEMENTS I_AnalogChannel_Standard
VAR
	Status : REFERENCE TO ST_AnalogInputStatus_EL30xx;
END_VAR

PROPERTY DataValid : BOOL
GET
DataValid := NOT Status.TxPDOState;
END_GET
END_PROPERTY

PROPERTY Error : BOOL
GET
Error := Status.Error;
END_GET
END_PROPERTY

(*FB_Init is always available implicitly and it is used primarily for initialization.
The return value is not evaluated. For a specific influence, you can also declare the
methods explicitly and provide additional code there with the standard initialization
code. You can evaluate the return value.*)
METHOD FB_Init : BOOL
VAR_INPUT
	(* TRUE: the retain variables are initialized (reset warm / reset cold)*)
	bInitRetains : BOOL;

	(* TRUE: the instance will be copied to the copy code afterward (online change)   *)
	bInCopyCode : BOOL;
	Name		: Core.T_MaxString;
	Input		: REFERENCE TO INT;
	Status		: REFERENCE TO ST_AnalogInputStatus_EL30xx;
END_VAR
THIS^.Status REF= Status;
END_METHOD

PROPERTY Limit1High : BOOL
GET
Limit1High := Status.Limit1H;
END_GET
END_PROPERTY

PROPERTY Limit1Low : BOOL
GET
Limit1Low := Status.Limit1L;
END_GET
END_PROPERTY

PROPERTY Limit2High : BOOL
GET
Limit2High := Status.Limit2H;
END_GET
END_PROPERTY

PROPERTY Limit2Low : BOOL
GET
Limit2Low := Status.Limit2L;
END_GET
END_PROPERTY

PROPERTY Overrange : BOOL
GET
Overrange := Status.Overrange;
END_GET
END_PROPERTY

PROPERTY Underrange : BOOL
GET
Underrange := Status.Underrrange;
END_GET
END_PROPERTY

END_FUNCTION_BLOCK

// Components/Analog/AnalogOutput
FUNCTION_BLOCK AnalogOutput EXTENDS Component IMPLEMENTS I_AnalogOutput, I_AnalogScalable, I_CalibratableLinear
VAR
	Output			 : REFERENCE TO INT;
	Forcible		 : ForcibleInt(_Name);
	_Scale			 : I_AnalogScale;
	_CalibrateLinear : I_CalibrateLinear;
	_CalibrateCustom : I_TransformLRealValue;
END_VAR

VAR
	{attribute 'hide'}
	DefaultScale : AnalogScale;
	{attribute 'hide'}
	DefaultCalibration : Calibrate;
END_VAR

PROPERTY CalibrateCustom : I_TransformLrealValue
SET
_CalibrateCustom := CalibrateCustom;
END_SET
END_PROPERTY

PROPERTY CalibrateLinear : I_CalibrateLinear
GET
CalibrateLinear := _CalibrateLinear;
END_GET
SET
_CalibrateLinear := CalibrateLinear;
END_SET
END_PROPERTY

(*FB_Init is always available implicitly and it is used primarily for initialization.
The return value is not evaluated. For a specific influence, you can also declare the
methods explicitly and provide additional code there with the standard initialization
code. You can evaluate the return value.*)
METHOD FB_Init : BOOL
VAR_INPUT
	(* TRUE: the retain variables are initialized (reset warm / reset cold)*)
	bInitRetains : BOOL;

	(* TRUE: the instance will be copied to the copy code afterward (online change)   *)
	bInCopyCode : BOOL;
	Name		: T_MaxString;
	Output		: REFERENCE TO INT;
END_VAR
_Scale			 := DefaultScale;
_CalibrateLinear := DefaultCalibration;
THIS^.Output	 REF= Output;
END_METHOD

{attribute 'monitoring' := 'call'}
PROPERTY Force : E_ForceState
GET
Force := Forcible.CurrentForceState;
END_GET
SET
VAR
	ForceString : T_MaxString := TO_STRING(Force);
END_VAR
Forcible.SetForceState(Force);
END_SET
END_PROPERTY

PROPERTY ForceValue : INT
GET
ForceValue := Forcible.ForceValue;
END_GET
SET
Forcible.ForceValue := ForceValue;
END_SET
END_PROPERTY

{attribute 'monitoring' := 'call'}
PROPERTY RawValue : INT
GET
RawValue := Output;
END_GET
SET
Forcible.Input := RawValue;
Output		   := Forcible.Output;
END_SET
END_PROPERTY

PROPERTY Scale : I_AnalogScale
GET
Scale := _Scale;
END_GET
SET
_Scale := Scale;
END_SET
END_PROPERTY

{attribute 'monitoring' := 'call'}
PROPERTY Value : LREAL
GET
IF _CalibrateCustom = 0 THEN
	Value := _CalibrateLinear.Transform(_Scale.Transform(RawValue));
ELSE
	Value := _CalibrateCustom.Transform(_Scale.Transform(RawValue));
END_IF
END_GET
SET
IF _CalibrateCustom = 0 THEN
	RawValue := LREAL_TO_INT(_Scale.Transform(_CalibrateLinear.Transform(Value, TRUE)));
ELSE
	RawValue := LREAL_TO_INT(_Scale.Transform(_CalibrateCustom.Transform(Value, TRUE)));
END_IF
END_SET
END_PROPERTY

END_FUNCTION_BLOCK

// Components/CoE/Interface/I_CoeAccess
INTERFACE I_CoeAccess EXTENDS I_Base

PROPERTY CoE : I_CoeDevice
GET
END_GET
END_PROPERTY

END_INTERFACE

// Components/CoE/Interface/I_CoeDevice
INTERFACE I_CoeDevice EXTENDS I_Component, I_TaskResult

PROPERTY AdsAddr : REFERENCE TO AMSADDR
GET
END_GET
SET
END_SET
END_PROPERTY

METHOD Read
VAR_INPUT
	Index	 : WORD;
	SubIndex : BYTE;
	pDstBuf	 : PVOID;
	BufLen	 : UDINT;
END_VAR
END_METHOD

METHOD Write
VAR_INPUT
	Index	 : WORD;
	SubIndex : BYTE;
	pDstBuf	 : PVOID;
	BufLen	 : UDINT;
END_VAR
END_METHOD

END_INTERFACE

// Components/CoE/CoeDevice
FUNCTION_BLOCK CoeDevice EXTENDS CyclicComponent IMPLEMENTS I_CoeDevice
VAR
	{attribute 'hide'}
	_Error : BOOL;
	{attribute 'hide'}
	_Busy : BOOL;
	{attribute 'hide'}
	_ErrorId : UDINT;
	_AdsAddr : REFERENCE TO AMSADDR;
	CoeRead	 : FB_EcCoESdoReadEx;
	CoeWrite : FB_EcCoESdoReadEx;
END_VAR

{attribute 'monitoring' := 'call'}
PROPERTY Busy : BOOL
GET
Busy := _Busy;
END_GET
END_PROPERTY

{attribute 'monitoring' := 'call'}
PROPERTY Error : BOOL
GET
Error := _Error;
END_GET
END_PROPERTY

{attribute 'monitoring' := 'call'}
PROPERTY ErrorId : UDINT
GET
ErrorID := _ErrorID;
END_GET
END_PROPERTY

PROPERTY AdsAddr : REFERENCE TO AMSADDR
GET
AdsAddr REF= _AdsAddr;
END_GET
SET
_AdsAddr REF= AdsAddr;
END_SET
END_PROPERTY

METHOD CyclicLogic
VAR_INST
END_VAR
IF NOT __ISVALIDREF(_AdsAddr) THEN
	RETURN;
END_IF

CoeRead(sNetId := F_CreateAmsNetId(AdsAddr.netId), nSlaveAddr := AdsAddr.port, tTimeout := T#1S);
CoeWrite(sNetId := F_CreateAmsNetId(AdsAddr.netId), nSlaveAddr := AdsAddr.port, tTimeout := T#1S);
CoeRead.bExecute  := FALSE;
CoeWrite.bExecute := FALSE;
_Busy			  := CoeRead.bBusy OR CoeWrite.bBusy;
_Error			  := CoeRead.bError OR CoeWrite.bError;
IF CoeRead.bError THEN
	_ErrorId := CoeRead.nErrId;
END_IF

IF CoeWrite.bError THEN
	_ErrorId := CoeWrite.nErrId;
END_IF
END_METHOD

METHOD Read
VAR_INPUT
	Index	 : WORD;
	SubIndex : BYTE;
	pDstBuf	 : PVOID;
	BufLen	 : UDINT;
END_VAR
IF _Busy THEN
	RETURN;
END_IF

CoeRead.nSubIndex		:= SubIndex;
CoeRead.nIndex			:= Index;
CoeRead.pDstBuf			:= pDstBuf;
CoeRead.cbBufLen		:= BufLen;
CoeRead.bCompleteAccess := SubIndex = 0;
_Busy					:= TRUE;
CoeRead.bExecute		:= TRUE;
END_METHOD

METHOD Write
VAR_INPUT
	Index	 : WORD;
	SubIndex : BYTE;
	pDstBuf	 : PVOID;
	BufLen	 : UDINT;
END_VAR
IF _Busy THEN
	RETURN;
END_IF

CoeWrite.nSubIndex		 := SubIndex;
CoeWrite.nIndex			 := Index;
CoeWrite.pDstBuf		 := pDstBuf;
CoeWrite.cbBufLen		 := BufLen;
CoeWrite.bCompleteAccess := SubIndex = 0;
_Busy					 := TRUE;
CoeWrite.bExecute		 := TRUE;
END_METHOD

END_FUNCTION_BLOCK

// Components/CoE/NullCoeDevice
FUNCTION_BLOCK NullCoeDevice EXTENDS CyclicComponent IMPLEMENTS I_CoeDevice
VAR
END_VAR

PROPERTY AdsAddr : REFERENCE TO AMSADDR
GET
END_GET
SET
END_SET
END_PROPERTY

{attribute 'monitoring' := 'call'}
PROPERTY Busy : BOOL
GET
END_GET
END_PROPERTY

METHOD CyclicLogic
END_METHOD

{attribute 'monitoring' := 'call'}
PROPERTY Error : BOOL
GET
END_GET
END_PROPERTY

{attribute 'monitoring' := 'call'}
PROPERTY ErrorId : UDINT
GET
END_GET
END_PROPERTY

METHOD Read
VAR_INPUT
	Index	 : WORD;
	SubIndex : BYTE;
	pDstBuf	 : PVOID;
	BufLen	 : UDINT;
END_VAR
END_METHOD

METHOD Write
VAR_INPUT
	Index	 : WORD;
	SubIndex : BYTE;
	pDstBuf	 : PVOID;
	BufLen	 : UDINT;
END_VAR
END_METHOD

END_FUNCTION_BLOCK

// Components/Cylinder/Interface/I_Cylinder
INTERFACE I_Cylinder EXTENDS I_CylinderCommand, I_CylinderStatus, I_Component, I_TaskResult, I_Resettable

{attribute 'monitoring' := 'call'}
PROPERTY ExtendTimeout : TIME
GET
END_GET
SET
END_SET
END_PROPERTY

{attribute 'monitoring' := 'call'}
PROPERTY RetractTimeout : TIME
GET
END_GET
SET
END_SET
END_PROPERTY

END_INTERFACE

// Components/Cylinder/Interface/I_CylinderCommand
INTERFACE I_CylinderCommand EXTENDS I_Base

METHOD Extend
END_METHOD

METHOD Retract
END_METHOD

END_INTERFACE

// Components/Cylinder/Interface/I_CylinderStatus
INTERFACE I_CylinderStatus EXTENDS I_Base

{attribute 'monitoring' := 'call'}
PROPERTY Extended : BOOL
GET
END_GET
END_PROPERTY

{attribute 'monitoring' := 'call'}
PROPERTY Extending : BOOL
GET
END_GET
END_PROPERTY

{attribute 'monitoring' := 'call'}
PROPERTY Retracted : BOOL
GET
END_GET
END_PROPERTY

{attribute 'monitoring' := 'call'}
PROPERTY Retracting : BOOL
GET
END_GET
END_PROPERTY

END_INTERFACE

// Components/Cylinder/Cylinder
FUNCTION_BLOCK Cylinder EXTENDS CyclicComponent IMPLEMENTS I_Cylinder
VAR
	ExtendOutput   : I_DigitalOutput;
	RetractOutput  : I_DigitalOutput;
	ExtendedInput  : I_DigitalInput;
	RetractedInput : I_DigitalInput;
	CylinderState  : E_CylinderState;
	{attribute 'hide'}
	_ExtendTimeout : TIME;
	{attribute 'hide'}
	_RetractTimeout : TIME;
	{attribute 'hide'}
	_Busy : BOOL;
	{attribute 'hide'}
	_Error : BOOL;
	{attribute 'hide'}
	_ErrorId : UDINT;
END_VAR

VAR
	{attribute 'hide'}
	NullEO : BOOL;
	{attribute 'hide'}
	NullExtendOutput : DigitalOutput('Null Digital Output', NullEO);
	{attribute 'hide'}
	NullRO : BOOL;
	{attribute 'hide'}
	NullRetractOutput : DigitalOutput('Null Digital Output', NullRO);
	{attribute 'hide'}
	NullEI : BOOL;
	{attribute 'hide'}
	NullExtendedInput : DigitalInput_NO('Null Digital Input', NullEI);
	{attribute 'hide'}
	NullRI : BOOL;
	{attribute 'hide'}
	NullRetractedInput : DigitalInput_NO('Null Digital Input', NullRI);
END_VAR

METHOD CyclicLogic
VAR_INST
	TON_RetractTimeout : TON;
	TON_ExtendTimeout  : TON;
END_VAR
NullEI := ExtendOutput.On;
NullRI := RetractOutput.On;
CASE CylinderState OF
	E_CylinderState.Undefined:
		IF ExtendedInput.IsActive THEN
			CylinderState := E_CylinderState.Extended;
		ELSIF RetractedInput.IsActive THEN
			CylinderState := E_CylinderState.Retracted;
		END_IF

	E_CylinderState.Extending:
		IF ExtendedInput.IsActive THEN
			CylinderState := E_CylinderState.Extended;
		END_IF

	E_CylinderState.Retracting:
		IF RetractedInput.IsActive THEN
			CylinderState := E_CylinderState.Retracted;
		END_IF
END_CASE

IF ExtendedInput.IsActive AND RetractedInput.IsActive THEN
	CylinderState := E_CylinderState.Undefined;
END_IF

// Generate Errors
IF CylinderState = E_CylinderState.Extending THEN
	IF _ExtendTimeout > T#0.0S THEN
		TON_ExtendTimeout(IN := TRUE, PT := _ExtendTimeout);
		IF TON_ExtendTimeout.Q THEN
			_Error	 := TRUE;
			_ErrorId := E_CylinderErrorId.ExtendTimeout;
		END_IF
	END_IF
ELSE
	TON_ExtendTimeout(IN := FALSE);
END_IF

IF CylinderState = E_CylinderState.Retracting THEN
	IF _RetractTimeout > T#0.0S THEN
		TON_RetractTimeout(IN := TRUE, PT := _RetractTimeout);
		IF TON_RetractTimeout.Q THEN
			_Error	 := TRUE;
			_ErrorId := E_CylinderErrorId.RetractTimeout;
		END_IF
	END_IF
ELSE
	TON_RetractTimeout(IN := FALSE);
END_IF

IF CylinderState = E_CylinderState.Extended THEN
	IF NOT ExtendedInput.IsActive THEN
		CylinderState := E_CylinderState.Undefined;
		_Error		  := TRUE;
		_ErrorId	  := E_CylinderErrorId.ExtendedPlausibility;
	END_IF
END_IF

IF CylinderState = E_CylinderState.Retracted THEN
	IF NOT RetractedInput.IsActive THEN
		CylinderState := E_CylinderState.Undefined;
		_Error		  := TRUE;
		_ErrorId	  := E_CylinderErrorId.RetractedPlausibility;
	END_IF
END_IF

IF ExtendedInput.IsActive AND RetractedInput.IsActive THEN
	CylinderState := E_CylinderState.Undefined;
	_Error		  := TRUE;
	_ErrorId	  := E_CylinderErrorId.BothSensorsActive;
END_IF

_Busy := (CylinderState = E_CylinderState.Extending) OR (CylinderState = E_CylinderState.Retracting);
END_METHOD

{attribute 'monitoring' := 'call'}
PROPERTY Busy : BOOL
GET
Busy := _Busy;
END_GET
END_PROPERTY

{attribute 'monitoring' := 'call'}
PROPERTY Error : BOOL
GET
Error := _Error;
END_GET
END_PROPERTY

{attribute 'monitoring' := 'call'}
PROPERTY ErrorId : UDINT
GET
ErrorID := _ErrorID;
END_GET
END_PROPERTY

METHOD Extend
IF CylinderState <> E_CylinderState.Extended THEN
	RetractOutput.On := FALSE;
	ExtendOutput.On	 := TRUE;
	CylinderState	 := E_CylinderState.Extending;
END_IF
END_METHOD

{attribute 'monitoring' := 'call'}
PROPERTY Extended : BOOL
GET
Extended := CylinderState = E_CylinderState.Extended;
END_GET
END_PROPERTY

{attribute 'monitoring' := 'call'}
PROPERTY Extending : BOOL
GET
Extending := CylinderState = E_CylinderState.Extending;
END_GET
END_PROPERTY

{attribute 'monitoring' := 'call'}
PROPERTY ExtendTimeout : TIME
GET
ExtendTimeout := _ExtendTimeout;
END_GET
SET
_ExtendTimeout := ExtendTimeout;
END_SET
END_PROPERTY

METHOD Retract
IF CylinderState <> E_CylinderState.Retracted THEN
	ExtendOutput.On	 := FALSE;
	RetractOutput.On := TRUE;
	CylinderState	 := E_CylinderState.Retracting;
END_IF
END_METHOD

{attribute 'monitoring' := 'call'}
PROPERTY Retracted : BOOL
GET
Retracted := CylinderState = E_CylinderState.Retracted;
END_GET
END_PROPERTY

{attribute 'monitoring' := 'call'}
PROPERTY Retracting : BOOL
GET
Retracting := CylinderState = E_CylinderState.Retracting;
END_GET
END_PROPERTY

{attribute 'monitoring' := 'call'}
PROPERTY RetractTimeout : TIME
GET
RetractTimeout := _RetractTimeout;
END_GET
SET
_RetractTimeout := RetractTimeout;
END_SET
END_PROPERTY

METHOD Reset
_Error	 := FALSE;
_ErrorId := 0;
END_METHOD

//FB_Init is always available implicitly and it is used primarily for initialization.

//The return value is not evaluated. For a specific influence, you can also declare the

//methods explicitly and provide additional code there with the standard initialization

//code. You can evaluate the return value.
METHOD FB_Init : BOOL
VAR_INPUT
	bInitRetains   : BOOL; // TRUE: the retain variables are initialized (reset warm / reset cold)
	bInCopyCode	   : BOOL; // TRUE: the instance will be copied to the copy code afterward (online change)  
	Name		   : T_MaxString;
	ExtendOutput   : I_DigitalOutput;
	RetractOutput  : I_DigitalOutput;
	ExtendedInput  : I_DigitalInput;
	RetractedInput : I_DigitalInput;
END_VAR
IF ExtendOutput = 0 THEN
	THIS^.ExtendOutput := NullExtendOutput;
ELSE
	THIS^.ExtendOutput := ExtendOutput;
END_IF

IF RetractOutput = 0 THEN
	THIS^.RetractOutput := NullRetractOutput;
ELSE
	THIS^.RetractOutput := RetractOutput;
END_IF

IF ExtendedInput = 0 THEN
	THIS^.ExtendedInput := NullExtendedInput;
ELSE
	THIS^.ExtendedInput := ExtendedInput;
END_IF

IF RetractedInput = 0 THEN
	THIS^.RetractedInput := NullRetractedInput;
ELSE
	THIS^.RetractedInput := RetractedInput;
END_IF
END_METHOD

END_FUNCTION_BLOCK

// Components/Digital/Interface/I_DigitalOutput
INTERFACE I_DigitalOutput EXTENDS I_Component, I_ForcibleBool

{attribute 'monitoring' := 'call'}
PROPERTY On : BOOL
GET
END_GET
SET
END_SET
END_PROPERTY

END_INTERFACE

// Utilities/Force/Interface/I_ForcibleBool
INTERFACE I_ForcibleBool EXTENDS I_Base

{attribute 'monitoring' := 'call'}
PROPERTY Force : E_ForceState
GET
END_GET
SET
END_SET
END_PROPERTY

END_INTERFACE

// Components/Digital/Interface/I_DigitalInput
INTERFACE I_DigitalInput EXTENDS I_Component, I_ForcibleBool

{attribute 'monitoring' := 'call'}
PROPERTY IsActive : BOOL
GET
END_GET
END_PROPERTY

END_INTERFACE

// Components/Digital/DigitalOutput
FUNCTION_BLOCK DigitalOutput EXTENDS Component IMPLEMENTS I_DigitalOutput
VAR
	Output		   : REFERENCE TO BOOL;
	ForcableOutput : ForcibleBool(_Name);
END_VAR

//FB_Init is always available implicitly and it is used primarily for initialization.

//The return value is not evaluated. For a specific influence, you can also declare the

//methods explicitly and provide additional code there with the standard initialization

//code. You can evaluate the return value.
METHOD FB_Init : BOOL
VAR_INPUT
	bInitRetains : BOOL; // TRUE: the retain variables are initialized (reset warm / reset cold)
	bInCopyCode	 : BOOL; // TRUE: the instance will be copied to the copy code afterward (online change)   
	Name		 : T_MaxString;
	Output		 : REFERENCE TO BOOL;
END_VAR
THIS^.Output REF= Output;
END_METHOD

{attribute 'monitoring' := 'call'}
PROPERTY Force : E_ForceState
GET
Force := ForcableOutput.CurrentForceState;
END_GET
SET
ForcableOutput.SetForceState(Force);
Output := ForcableOutput.Output;
END_SET
END_PROPERTY

{attribute 'monitoring' := 'call'}
PROPERTY On : BOOL
GET
On := Output;
END_GET
SET
ForcableOutput.Input := On;
Output				 := ForcableOutput.Output;
END_SET
END_PROPERTY

END_FUNCTION_BLOCK

// Utilities/Force/ForcibleBool
FUNCTION_BLOCK ForcibleBool
VAR
	Name			   : T_MaxString;
	_CurrentForceState : E_ForceState;
	ForceEvent		   : FB_TcAlarm;
	RequestedState	   : BOOL;
	_Output			   : BOOL;
END_VAR

METHOD PRIVATE ResolveOutput
VAR
	ForceString : T_MaxString := TO_STRING(_CurrentForceState);
END_VAR
CASE _CurrentForceState OF
	E_ForceState.Unforced:
		_Output := RequestedState;
		ForceEvent.Clear();

	E_ForceState.ForceOn:
		IF NOT ForceEvent.bActive THEN
			ForceEvent.ipArguments.Clear().AddString(Name).AddString(ForceString);
			ForceEvent.Raise();
		END_IF

		_Output := TRUE;

	E_ForceState.ForceOff:
		IF NOT ForceEvent.bActive THEN
			ForceEvent.ipArguments.Clear().AddString(Name).AddString(ForceString);
			ForceEvent.Raise();
		END_IF

		_Output := FALSE;
END_CASE
END_METHOD

{attribute 'monitoring' := 'call'}
PROPERTY CurrentForceState : E_ForceState
GET
CurrentForceState := _CurrentForceState;
END_GET
END_PROPERTY

//FB_Init is always available implicitly and it is used primarily for initialization.

//The return value is not evaluated. For a specific influence, you can also declare the

//methods explicitly and provide additional code there with the standard initialization

//code. You can evaluate the return value.
METHOD FB_Init : BOOL
VAR_INPUT
	bInitRetains : BOOL; // TRUE: the retain variables are initialized (reset warm / reset cold)
	bInCopyCode	 : BOOL; // TRUE: the instance will be copied to the copy code afterward (online change) 
	Name		 : T_MaxString;
END_VAR
THIS^.Name := Name;
{analysis -15}
IF NOT ForceEvent.EqualsToEventEntryEx(TC_EVENTS.IO.ForceActive) THEN
	ForceEvent.CreateEx(TC_EVENTS.IO.ForceActive, 0);
END_IF
END_METHOD

{attribute 'monitoring' := 'call'}
PROPERTY Input : BOOL
SET
RequestedState := Input;
ResolveOutput();
END_SET
END_PROPERTY

{attribute 'monitoring' := 'call'}
PROPERTY Output : BOOL
GET
Output := _Output;
END_GET
END_PROPERTY

METHOD SetForceState
VAR_INPUT
	ForceState : E_ForceState;
END_VAR
IF ForceState = _CurrentForceState THEN
	RETURN;
END_IF

_CurrentForceState := ForceState;
ResolveOutput();
END_METHOD

END_FUNCTION_BLOCK

// Components/Digital/DigitalInput_NO
FUNCTION_BLOCK DigitalInput_NO EXTENDS Component IMPLEMENTS I_DigitalInput
VAR
	Input		  : REFERENCE TO BOOL;
	ForcibleInput : ForcibleBool(_Name);
END_VAR

//FB_Init is always available implicitly and it is used primarily for initialization.

//The return value is not evaluated. For a specific influence, you can also declare the

//methods explicitly and provide additional code there with the standard initialization

//code. You can evaluate the return value.
METHOD FB_Init : BOOL
VAR_INPUT
	bInitRetains : BOOL; // TRUE: the retain variables are initialized (reset warm / reset cold)
	bInCopyCode	 : BOOL; // TRUE: the instance will be copied to the copy code afterward (online change)   
	Name		 : T_MaxString;
	Input		 : REFERENCE TO BOOL;
END_VAR
THIS^.Input REF= Input;
END_METHOD

{attribute 'monitoring' := 'call'}
PROPERTY Force : E_ForceState
GET
Force := ForcibleInput.CurrentForceState;
END_GET
SET
VAR
	ForceString : T_MaxString := TO_STRING(Force);
END_VAR
ForcibleInput.SetForceState(Force);
END_SET
END_PROPERTY

{attribute 'monitoring' := 'call'}
PROPERTY IsActive : BOOL
GET
ForcibleInput.Input := Input;
IsActive			:= ForcibleInput.Output;
END_GET
END_PROPERTY

END_FUNCTION_BLOCK

// Components/Cylinder/Cylinder_HMI
FUNCTION_BLOCK Cylinder_HMI EXTENDS HmiFunction
VAR
	Cylinder : I_Cylinder;
	{ attribute 'TcHmiSymbol.AddSymbol' }
	{ attribute 'TcHmiSymbol.AddSymbol.UserGroups' := '__SystemAdministrators,Admin' }
	Cylinder_HMI : ST_Cylinder_HMI;
END_VAR

PROPERTY ExtendPermissive : I_Permissive
GET
ExtendPermissive := Cylinder_HMI.Extend.Permissive;
END_GET
END_PROPERTY

PROPERTY RetractPermissive : I_Permissive
GET
RetractPermissive := Cylinder_HMI.Retract.Permissive;
END_GET
END_PROPERTY

PROPERTY ControlObject : I_Base
SET
__QueryInterface(ControlObject,Cylinder);
END_SET
END_PROPERTY

METHOD CyclicLogic
VAR_INST
	ExtendRT  : R_TRIG;
	RetractRT : R_TRIG;
END_VAR
IF Cylinder = 0 THEN
	RETURN;
END_IF

Cylinder_HMI.HmiEnabled := Enabled;
Cylinder_HMI.Name		:= Cylinder.Name;
Cylinder_HMI.Busy		:= Cylinder.Busy;
Cylinder_HMI.Error		:= Cylinder.Error;
Cylinder_HMI.ErrorId	:= Cylinder.ErrorId;
Cylinder_HMI.Extended	:= Cylinder.Extended;
Cylinder_HMI.Retracted	:= Cylinder.Retracted;
// HMI Commands
IF Enabled THEN
	ExtendRT(CLK := Cylinder_HMI.Extend.Active);
	IF ExtendRT.Q THEN
		IF Cylinder_HMI.Extend.Permissive.OK THEN
			Cylinder.Extend();
		END_IF
	END_IF

	RetractRT(CLK := Cylinder_HMI.Retract.Active);
	IF RetractRT.Q THEN
		IF Cylinder_HMI.Retract.Permissive.OK THEN
			Cylinder.Retract();
		END_IF
	END_IF
END_IF
END_METHOD

PROPERTY ExtendCommandName : STRING
GET
ExtendCommandName := Cylinder_HMI.Extend.Name;
END_GET
SET
Cylinder_HMI.Extend.Name := ExtendCommandName;
END_SET
END_PROPERTY

PROPERTY ExtendedName : STRING
GET
ExtendedName := Cylinder_HMI.ExtendedName;
END_GET
SET
Cylinder_HMI.ExtendedName := ExtendedName;
END_SET
END_PROPERTY

(*FB_Init is always available implicitly and it is used primarily for initialization.
The return value is not evaluated. For a specific influence, you can also declare the
methods explicitly and provide additional code there with the standard initialization
code. You can evaluate the return value.*)
METHOD FB_Init : BOOL
VAR_INPUT
	(* TRUE: the retain variables are initialized (reset warm / reset cold)*)
	bInitRetains : BOOL;

	(* TRUE: the instance will be copied to the copy code afterward (online change)   *)
	bInCopyCode : BOOL;
	Name		: Core.T_MaxString;
	Cylinder	: I_Cylinder;
END_VAR
THIS^.Cylinder := Cylinder;
ControlType	   := 'Cylinder';
LinkObject	   := 'Cylinder_HMI';
END_METHOD

PROPERTY RetractCommandName : STRING
GET
RetractCommandName := Cylinder_HMI.Retract.Name;
END_GET
SET
Cylinder_HMI.Retract.Name := RetractCommandName;
END_SET
END_PROPERTY

PROPERTY RetractedName : STRING
GET
RetractedName := Cylinder_HMI.RetractedName;
END_GET
SET
Cylinder_HMI.RetractedName := RetractedName;
END_SET
END_PROPERTY

END_FUNCTION_BLOCK

// Components/Cylinder/Cylinder_TcEvents
FUNCTION_BLOCK Cylinder_TcEvents EXTENDS CyclicComponent IMPLEMENTS I_EventReactionTcEvents
VAR
	Cylinder : I_Cylinder;
	Events	 : TcEventClass(CONCAT(Name, ' Events'));
END_VAR

METHOD GetHighestActiveEventReaction : DINT
GetHighestActiveEventReaction := Events.GetHighestActiveEventReaction();
END_METHOD

METHOD GetHighestActiveEventSeverity : Core.TcEventSeverity
GetHighestActiveEventSeverity := Events.GetHighestActiveEventSeverity();
END_METHOD

METHOD Reset
Events.Reset();
END_METHOD

METHOD SetEventReactions
VAR_INPUT
	Verbose	 : DINT := 0;
	Info	 : DINT := 1;
	Warning	 : DINT := 2;
	Error	 : DINT := 3;
	Critical : DINT := 4;
END_VAR
Events.SetEventReactions(Verbose,
						 Info,
						 Warning,
						 Error,
						 Critical);
END_METHOD

METHOD CyclicLogic
IF Cylinder.Error THEN
	CASE Cylinder.ErrorId OF
		E_CylinderErrorId.NoError:
			;

		E_CylinderErrorId.BothSensorsActive:
			Events.RaiseEvent(E_cylinder.BothSensorsActive);

		E_CylinderErrorId.ExtendedPlausibility:
			Events.RaiseEvent(E_cylinder.ExtendedPlausibility);

		E_CylinderErrorId.ExtendTimeout:
			Events.RaiseEvent(E_cylinder.ExtendTimeout);

		E_CylinderErrorId.RetractedPlausibility:
			Events.RaiseEvent(E_cylinder.RetractedPlausibility);

		E_CylinderErrorId.RetractTimeout:
			Events.RaiseEvent(E_cylinder.RetractTimeout);
	END_CASE
END_IF
END_METHOD

(*FB_Init is always available implicitly and it is used primarily for initialization.
The return value is not evaluated. For a specific influence, you can also declare the
methods explicitly and provide additional code there with the standard initialization
code. You can evaluate the return value.*)
METHOD FB_Init : BOOL
VAR_INPUT
	(* TRUE: the retain variables are initialized (reset warm / reset cold)*)
	bInitRetains : BOOL;

	(* TRUE: the instance will be copied to the copy code afterward (online change)   *)
	bInCopyCode : BOOL;
	Name		: Core.T_MaxString;
	Cylinder	: I_Cylinder;
END_VAR
THIS^.Cylinder := Cylinder;
Events.GenerateTcEvents(Cylinder.Name, ADR(TC_events.Cylinder), SIZEOF(ST_Cylinder));
END_METHOD

END_FUNCTION_BLOCK

// Components/Digital/Visitor/ForceVisitor
FUNCTION_BLOCK ForceVisitor IMPLEMENTS I_ComponentVisitor
VAR
	Forcible : I_ForcibleBool;
	{attribute 'hide'}
	_ForceState : E_ForceState;
END_VAR

{attribute 'monitoring' := 'call'}
PROPERTY Force : E_ForceState
GET
Force := _ForceState;
END_GET
SET
_ForceState := Force;
END_SET
END_PROPERTY

METHOD VisitComponent
VAR_INPUT
	Component : Core.I_Component;
END_VAR
IF __QUERYINTERFACE(Component, Forcible) THEN
	Forcible.Force := Force;
END_IF
END_METHOD

END_FUNCTION_BLOCK

// Components/Digital/Visitor/ReleaseAllForceVisitor
FUNCTION_BLOCK ReleaseAllForceVisitor IMPLEMENTS I_ModuleVisitor, I_ComponentVisitor
VAR
END_VAR

METHOD ReleaseForces : BOOL;
VAR_INPUT
	Module : I_Module;
END_VAR
Module.Accept(THIS^);
END_METHOD

METHOD VisitComponent
VAR_INPUT
	Component : Core.I_Component;
END_VAR

VAR_INST
	Forcible : I_ForcibleBool;
END_VAR
IF __QUERYINTERFACE(Component, Forcible) THEN
	Forcible.Force := E_ForceState.Unforced;
END_IF
END_METHOD

METHOD VisitModule
VAR_INPUT
	Module : Core.I_Module;
END_VAR
Module.Components.Accept(THIS^);
Module.Modules.Accept(THIS^);
END_METHOD

END_FUNCTION_BLOCK

// Components/Digital/DigitalInput_Combiner
FUNCTION_BLOCK DigitalInput_Combiner
VAR_GENERIC CONSTANT
	NumberOfCombinedInputs : DINT := 2;
END_VAR
EXTENDS Component IMPLEMENTS I_DigitalInput
VAR
	Inputs : ARRAY[0..(NumberOfCombinedInputs - 1)] OF I_DigitalInput;
	{attribute 'hide'}
	_Force : E_ForceState;
END_VAR

METHOD AddInput
VAR_INPUT
	Input : I_DigitalInput;
END_VAR

VAR
	i : DINT;
END_VAR
FOR i := 0 TO (NumberOfCombinedInputs - 1) DO
	IF Inputs[i] = Input THEN
		RETURN;
	END_IF
END_FOR

FOR i := 0 TO (NumberOfCombinedInputs - 1) DO
	IF Inputs[i] = 0 THEN
		Inputs[i] := Input;
		RETURN;
	END_IF
END_FOR
END_METHOD

{attribute 'monitoring' := 'call'}
PROPERTY Force : E_ForceState
GET
Force := _Force;
END_GET
SET
VAR
	i : DINT;
END_VAR
_Force := Force;
IF Inputs[0] = 0 THEN
	RETURN;
END_IF

FOR i := 0 TO (NumberOfCombinedInputs - 1) DO
	IF Inputs[i] = 0 THEN
		RETURN;
	END_IF

	Inputs[i].Force := Force;
END_FOR
END_SET
END_PROPERTY

{attribute 'monitoring' := 'call'}
PROPERTY IsActive : BOOL
GET
VAR
	i : DINT;
END_VAR
IF Inputs[0] = 0 THEN
	RETURN;
END_IF

IsActive := TRUE;
FOR i := 0 TO (NumberOfCombinedInputs - 1) DO
	IF Inputs[i] = 0 THEN
		RETURN;
	END_IF

	IsActive := IsActive AND Inputs[i].IsActive;
END_FOR
END_GET
END_PROPERTY

END_FUNCTION_BLOCK

// Components/Digital/DigitalInput_DebounceFallingEdge
FUNCTION_BLOCK DigitalInput_DebounceFallingEdge EXTENDS CyclicComponent IMPLEMENTS I_DigitalInput
VAR
	Input : I_DigitalInput;
	{attribute 'hide'}
	_DebounceTime		: TIME;
	DebounceFallingEdge : TOF;
END_VAR

METHOD CyclicLogic
DebounceFallingEdge(IN := Input.IsActive, PT := _DebounceTime);
END_METHOD

{attribute 'monitoring' := 'call'}
PROPERTY DebounceTime : TIME
GET
DebounceTime := _DebounceTime;
END_GET
SET
_DebounceTime := DebounceTime;
END_SET
END_PROPERTY

(*FB_Init is always available implicitly and it is used primarily for initialization.
The return value is not evaluated. For a specific influence, you can also declare the
methods explicitly and provide additional code there with the standard initialization
code. You can evaluate the return value.*)
METHOD FB_Init : BOOL
VAR_INPUT
	(* TRUE: the retain variables are initialized (reset warm / reset cold)*)
	bInitRetains : BOOL;

	(* TRUE: the instance will be copied to the copy code afterward (online change)   *)
	bInCopyCode : BOOL;
	Name		: Core.T_MaxString;
	Input		: I_DigitalInput;
END_VAR
THIS^.Input := Input;
END_METHOD

{attribute 'monitoring' := 'call'}
PROPERTY Force : E_ForceState
GET
Force := Input.Force;
END_GET
SET
Input.Force := Force;
END_SET
END_PROPERTY

{attribute 'monitoring' := 'call'}
PROPERTY IsActive : BOOL
GET
IsActive := DebounceFallingEdge.Q;
END_GET
END_PROPERTY

END_FUNCTION_BLOCK

// Components/Digital/DigitalInput_DebounceRisingEdge
FUNCTION_BLOCK DigitalInput_DebounceRisingEdge EXTENDS CyclicComponent IMPLEMENTS I_DigitalInput
VAR
	Input : I_DigitalInput;
	{attribute 'hide'}
	_DebounceTime	   : TIME;
	DebounceRisingEdge : TON;
END_VAR

METHOD CyclicLogic
DebounceRisingEdge(IN := Input.IsActive, PT := _DebounceTime);
END_METHOD

{attribute 'monitoring' := 'call'}
PROPERTY DebounceTime : TIME
GET
DebounceTime := _DebounceTime;
END_GET
SET
_DebounceTime := DebounceTime;
END_SET
END_PROPERTY

(*FB_Init is always available implicitly and it is used primarily for initialization.
The return value is not evaluated. For a specific influence, you can also declare the
methods explicitly and provide additional code there with the standard initialization
code. You can evaluate the return value.*)
METHOD FB_Init : BOOL
VAR_INPUT
	(* TRUE: the retain variables are initialized (reset warm / reset cold)*)
	bInitRetains : BOOL;

	(* TRUE: the instance will be copied to the copy code afterward (online change)   *)
	bInCopyCode : BOOL;
	Name		: Core.T_MaxString;
	Input		: I_DigitalInput;
END_VAR
THIS^.Input := Input;
END_METHOD

{attribute 'monitoring' := 'call'}
PROPERTY Force : E_ForceState
GET
Force := Input.Force;
END_GET
SET
Input.Force := Force;
END_SET
END_PROPERTY

{attribute 'monitoring' := 'call'}
PROPERTY IsActive : BOOL
GET
IsActive := DebounceRisingEdge.Q;
END_GET
END_PROPERTY

END_FUNCTION_BLOCK

// Components/Digital/DigitalInput_HMI
FUNCTION_BLOCK DigitalInput_HMI EXTENDS HmiFunction
VAR
	DigitalInput : I_DigitalInput;
	{ attribute 'TcHmiSymbol.AddSymbol' }
	{ attribute 'TcHmiSymbol.AddSymbol.UserGroups' := '__SystemAdministrators,Admin' }
	DigitalInput_HMI : ST_DigitalInput_HMI;
END_VAR

PROPERTY ControlObject : I_Base
SET
__QueryInterface(ControlObject,DigitalInput);
END_SET
END_PROPERTY

METHOD CyclicLogic
IF DigitalInput = 0 THEN
	RETURN;
END_IF

DigitalInput_HMI.Name		:= DigitalInput.Name;
DigitalInput_HMI.Active		:= DigitalInput.IsActive;
DigitalInput_HMI.HmiEnabled := Enabled;
IF Enabled THEN
	DigitalInput.Force := DigitalInput_HMI.Force;
END_IF
END_METHOD

(*FB_Init is always available implicitly and it is used primarily for initialization.
The return value is not evaluated. For a specific influence, you can also declare the
methods explicitly and provide additional code there with the standard initialization
code. You can evaluate the return value.*)
METHOD FB_Init : BOOL
VAR_INPUT
	(* TRUE: the retain variables are initialized (reset warm / reset cold)*)
	bInitRetains : BOOL;

	(* TRUE: the instance will be copied to the copy code afterward (online change)   *)
	bInCopyCode	 : BOOL;
	Name		 : Core.T_MaxString;
	DigitalInput : I_DigitalInput;
END_VAR
THIS^.DigitalInput := DigitalInput;
ControlType		   := 'DigitalInput';
LinkObject		   := 'DigitalInput_HMI';
END_METHOD

END_FUNCTION_BLOCK

// Components/Digital/DigitalInput_NC
FUNCTION_BLOCK DigitalInput_NC EXTENDS Component IMPLEMENTS I_DigitalInput
VAR
	Input		  : REFERENCE TO BOOL;
	ForcibleInput : ForcibleBool(_Name);
END_VAR

//FB_Init is always available implicitly and it is used primarily for initialization.

//The return value is not evaluated. For a specific influence, you can also declare the

//methods explicitly and provide additional code there with the standard initialization

//code. You can evaluate the return value.
METHOD FB_Init : BOOL
VAR_INPUT
	bInitRetains : BOOL; // TRUE: the retain variables are initialized (reset warm / reset cold)
	bInCopyCode	 : BOOL; // TRUE: the instance will be copied to the copy code afterward (online change)   
	Name		 : T_MaxString;
	Input		 : REFERENCE TO BOOL;
END_VAR
THIS^.Input REF= Input;
END_METHOD

{attribute 'monitoring' := 'call'}
PROPERTY Force : E_ForceState
GET
Force := ForcibleInput.CurrentForceState;
END_GET
SET
VAR
	ForceString : T_MaxString := TO_STRING(Force);
END_VAR
ForcibleInput.SetForceState(Force);
END_SET
END_PROPERTY

{attribute 'monitoring' := 'call'}
PROPERTY IsActive : BOOL
GET
ForcibleInput.Input := NOT Input;
IsActive			:= ForcibleInput.Output;
END_GET
END_PROPERTY

END_FUNCTION_BLOCK

// Components/Digital/DigitalOutput_HMI
FUNCTION_BLOCK DigitalOutput_HMI EXTENDS HmiFunction
VAR
	DigitalOutput : I_DigitalOutput;
	{ attribute 'TcHmiSymbol.AddSymbol' }
	{ attribute 'TcHmiSymbol.AddSymbol.UserGroups' := '__SystemAdministrators,Admin' }
	DigitalOutput_HMI : ST_DigitalOutput_HMI;
END_VAR

PROPERTY ControlObject : I_Base
SET
__QueryInterface(ControlObject,DigitalOutput);
END_SET
END_PROPERTY

METHOD CyclicLogic
IF DigitalOutput = 0 THEN
	RETURN;
END_IF

DigitalOutput_HMI.Name		 := DigitalOutput.Name;
DigitalOutput_HMI.On		 := DigitalOutput.On;
DigitalOutput_HMI.HmiEnabled := Enabled;
IF Enabled THEN
	DigitalOutput.Force := DigitalOutput_HMI.Force;
END_IF
END_METHOD

(*FB_Init is always available implicitly and it is used primarily for initialization.
The return value is not evaluated. For a specific influence, you can also declare the
methods explicitly and provide additional code there with the standard initialization
code. You can evaluate the return value.*)
METHOD FB_Init : BOOL
VAR_INPUT
	(* TRUE: the retain variables are initialized (reset warm / reset cold)*)
	bInitRetains : BOOL;

	(* TRUE: the instance will be copied to the copy code afterward (online change)   *)
	bInCopyCode	  : BOOL;
	Name		  : Core.T_MaxString;
	DigitalOutput : I_DigitalOutput;
END_VAR
THIS^.DigitalOutput := DigitalOutput;
ControlType			:= 'DigitalOutput';
LinkObject			:= 'DigitalOutput_HMI';
END_METHOD

END_FUNCTION_BLOCK

// Components/EtherCat/Interface/I_EcIoDevice
INTERFACE I_EcIoDevice EXTENDS I_IoDevice, I_CoeAccess

{attribute 'monitoring' := 'call'}
PROPERTY Bootstrap : BOOL
GET
END_GET
END_PROPERTY

PROPERTY Configuration : REFERENCE TO ST_EcSlaveConfigData
GET
END_GET
SET
END_SET
END_PROPERTY

{attribute 'monitoring' := 'call'}
PROPERTY DeviceError : BOOL
GET
END_GET
END_PROPERTY

{attribute 'monitoring' := 'call'}
PROPERTY Disabled : BOOL
GET
END_GET
END_PROPERTY

{attribute 'monitoring' := 'call'}
PROPERTY Init : BOOL
GET
END_GET
END_PROPERTY

{attribute 'monitoring' := 'call'}
PROPERTY InitCmdError : BOOL
GET
END_GET
END_PROPERTY

{attribute 'monitoring' := 'call'}
PROPERTY InvalidVPRS : BOOL
GET
END_GET
END_PROPERTY

{attribute 'monitoring' := 'call'}
PROPERTY OP : BOOL
GET
END_GET
END_PROPERTY

{attribute 'monitoring' := 'call'}
PROPERTY PreOp : BOOL
GET
END_GET
END_PROPERTY

{attribute 'monitoring' := 'call'}
PROPERTY SafeOp : BOOL
GET
END_GET
END_PROPERTY

PROPERTY State : REFERENCE TO ST_EcSlaveState
GET
END_GET
SET
END_SET
END_PROPERTY

END_INTERFACE

// Components/EtherCat/Interface/I_IoDevice
INTERFACE I_IoDevice EXTENDS I_Base

{attribute 'monitoring' := 'call'}
PROPERTY IoDataValid : BOOL
GET
END_GET
END_PROPERTY

END_INTERFACE

// Components/EtherCat/Interface/I_EtherCatDiagnosticEventProvider
INTERFACE I_EtherCatDiagnosticEventProvider EXTENDS I_EventReactionTcEvents

METHOD RaiseEtherCatDiagnosticEvent
VAR_INPUT
	EventId	  : UDINT;
	Argument1 : STRING := '';
	Argument2 : STRING := '';
	Argument3 : STRING := '';
END_VAR
END_METHOD

METHOD RaiseSyncUnitEvent
VAR_INPUT
	EventId	  : UDINT;
	Argument1 : STRING := '';
	Argument2 : STRING := '';
	Argument3 : STRING := '';
END_VAR
END_METHOD

END_INTERFACE

// Components/EtherCat/Interface/I_EtherCatMasterDiagnostic
INTERFACE I_EtherCatMasterDiagnostic EXTENDS I_Component, I_Resettable

{attribute 'monitoring' := 'call'}
PROPERTY ConfiguredSlaveCount : UINT
GET
END_GET
END_PROPERTY

METHOD GetIoDeviceByAddr : I_EcIoDevice
VAR_INPUT
	Addr : WORD;
END_VAR
END_METHOD

METHOD GetIoDeviceByName : I_EcIoDevice
VAR_INPUT
	Name : STRING(31);
END_VAR
END_METHOD

{attribute 'monitoring' := 'call'}
PROPERTY LocalAmsNetId : T_AmsNetId
GET
END_GET
END_PROPERTY

{attribute 'monitoring' := 'call'}
PROPERTY MasterAmsNetId : T_AmsNetId
GET
END_GET
END_PROPERTY

METHOD RegisterEventProvider
VAR_INPUT
	EventProvider : I_EtherCatDiagnosticEventProvider;
END_VAR
END_METHOD

{attribute 'monitoring' := 'call'}
PROPERTY SlaveCount : UINT
GET
END_GET
END_PROPERTY

END_INTERFACE

// Components/EtherCat/Interface/I_SyncUnitTask
INTERFACE I_SyncUnitTask EXTENDS I_Component

{attribute 'monitoring' := 'call'}
PROPERTY IoDataValid : BOOL
GET
END_GET
END_PROPERTY

{attribute 'monitoring' := 'call'}
PROPERTY IsHotConnect : BOOL
GET
END_GET
END_PROPERTY

{attribute 'monitoring' := 'call'}
PROPERTY PUBLIC SlaveCount : UINT
GET
END_GET
END_PROPERTY

END_INTERFACE

// Components/EtherCat/EtherCatIoDevice
FUNCTION_BLOCK EtherCatIoDevice EXTENDS CyclicComponent IMPLEMENTS I_EcIoDevice
VAR
	_Config	  : REFERENCE TO ST_EcSlaveConfigData;
	_State	  : REFERENCE TO ST_EcSlaveState;
	_SyncUnit : I_SyncUnitTask;
	_AmsAddr  : AMSADDR;
	CoeDevice : CoeDevice('CoE Terminal');
	{attribute 'hide'}
	NullCoeDevice : NullCoeDevice('Null Terminal');
END_VAR

{attribute 'monitoring' := 'call'}
PROPERTY Bootstrap : BOOL
GET
VAR
	DiagByte	: BYTE;
	BitMaskDiag : BYTE := 16#0F;
END_VAR
IF __ISVALIDREF(_State) THEN
	BitMaskDiag := 16#0F;
	DiagByte	:= _State.deviceState AND BitMaskDiag;
	Bootstrap	:= DiagByte = EC_DEVICE_STATE_BOOTSTRAP;
END_IF
END_GET
END_PROPERTY

PROPERTY CoE : I_CoeDevice
GET
IF _Config.nMailboxInSize = 0 THEN
	CoE := NullCoeDevice;
ELSE
	_AmsAddr.port	  := _Config.nAddr;
	CoeDevice.AdsAddr REF= _AmsAddr;
	CoE				  := CoeDevice;
END_IF
END_GET
SET
END_SET
END_PROPERTY

PROPERTY Configuration : REFERENCE TO ST_EcSlaveConfigData
GET
Configuration REF= _Config;
END_GET
SET
_Config REF= Configuration;
END_SET
END_PROPERTY

{attribute 'monitoring' := 'call'}
PROPERTY DeviceError : BOOL
GET
VAR
	DiagByte	: BYTE;
	BitMaskDiag : BYTE := 16#0F;
END_VAR
IF __ISVALIDREF(_State) THEN
	BitMaskDiag := 16#0F;
	DiagByte	:= _State.deviceState AND BitMaskDiag;
	DeviceError := DiagByte = EC_DEVICE_STATE_ERROR;
END_IF
END_GET
END_PROPERTY

{attribute 'monitoring' := 'call'}
PROPERTY Disabled : BOOL
GET
VAR
	DiagByte	: BYTE;
	BitMaskDiag : BYTE := 16#0F;
END_VAR
IF __ISVALIDREF(_State) THEN
	BitMaskDiag := 16#0F;
	DiagByte	:= _State.deviceState AND BitMaskDiag;
	Disabled	:= DiagByte = EC_DEVICE_STATE_DISABLED;
END_IF
END_GET
END_PROPERTY

{attribute 'monitoring' := 'call'}
PROPERTY Init : BOOL
GET
VAR
	DiagByte	: BYTE;
	BitMaskDiag : BYTE := 16#0F;
END_VAR
IF __ISVALIDREF(_State) THEN
	BitMaskDiag := 16#0F;
	DiagByte	:= _State.deviceState AND BitMaskDiag;
	Init		:= DiagByte = EC_DEVICE_STATE_INIT;
END_IF
END_GET
END_PROPERTY

{attribute 'monitoring' := 'call'}
PROPERTY InitCmdError : BOOL
GET
VAR
	DiagByte	: BYTE;
	BitMaskDiag : BYTE := 16#0F;
END_VAR
IF __ISVALIDREF(_State) THEN
	BitMaskDiag	 := 16#0F;
	DiagByte	 := _State.deviceState AND BitMaskDiag;
	InitCmdError := DiagByte = EC_DEVICE_STATE_INVALID_VPRS;
END_IF
END_GET
END_PROPERTY

{attribute 'monitoring' := 'call'}
PROPERTY InvalidVPRS : BOOL
GET
VAR
	DiagByte	: BYTE;
	BitMaskDiag : BYTE := 16#0F;
END_VAR
IF __ISVALIDREF(_State) THEN
	BitMaskDiag := 16#0F;
	DiagByte	:= _State.deviceState AND BitMaskDiag;
	InvalidVPRS := DiagByte = EC_DEVICE_STATE_INVALID_VPRS;
END_IF
END_GET
END_PROPERTY

{attribute 'monitoring' := 'call'}
PROPERTY IoDataValid : BOOL
GET
IF _SyncUnit <> 0 THEN
	IoDataValid := _SyncUnit.IoDataValid;
ELSE
	IoDataValid := TRUE;
END_IF
END_GET
END_PROPERTY

{attribute 'monitoring' := 'call'}
PROPERTY OP : BOOL
GET
VAR
	DiagByte	: BYTE;
	BitMaskDiag : BYTE := 16#0F;
END_VAR
IF __ISVALIDREF(_State) THEN
	BitMaskDiag := 16#0F;
	DiagByte	:= _State.deviceState AND BitMaskDiag;
	OP			:= DiagByte = EC_DEVICE_STATE_OP;
END_IF
END_GET
END_PROPERTY

{attribute 'monitoring' := 'call'}
PROPERTY PreOp : BOOL
GET
VAR
	DiagByte	: BYTE;
	BitMaskDiag : BYTE := 16#0F;
END_VAR
IF __ISVALIDREF(_State) THEN
	BitMaskDiag := 16#0F;
	DiagByte	:= _State.deviceState AND BitMaskDiag;
	PreOp		:= DiagByte = EC_DEVICE_STATE_PREOP;
END_IF
END_GET
END_PROPERTY

{attribute 'monitoring' := 'call'}
PROPERTY SafeOp : BOOL
GET
VAR
	DiagByte	: BYTE;
	BitMaskDiag : BYTE := 16#0F;
END_VAR
IF __ISVALIDREF(_State) THEN
	BitMaskDiag := 16#0F;
	DiagByte	:= _State.deviceState AND BitMaskDiag;
	SafeOp		:= DiagByte = EC_DEVICE_STATE_SAFEOP;
END_IF
END_GET
END_PROPERTY

PROPERTY State : REFERENCE TO ST_EcSlaveState
GET
State REF= _State;
END_GET
SET
_State REF= State;
END_SET
END_PROPERTY

PROPERTY AmsNetId : AMSNETID
SET
_AmsAddr.netId := AmsNetId;
END_SET
END_PROPERTY

METHOD CyclicLogic
IF _AmsAddr.port = 0 THEN
	_AmsAddr.port	  := _Config.nAddr;
	CoeDevice.AdsAddr REF= _AmsAddr;
END_IF

IF _Config.nMailboxInSize <> 0 THEN
	CoeDevice.CyclicLogic();
END_IF
END_METHOD

PROPERTY SyncUnit : I_SyncUnitTask
SET
_SyncUnit := SyncUnit;
END_SET
END_PROPERTY

END_FUNCTION_BLOCK

// Components/EtherCat/EtherCatMaster
FUNCTION_BLOCK EtherCatMaster
VAR_GENERIC CONSTANT
	FRAMES	   : UINT := 1;
	SYNC_UNITS : UINT := 2;
END_VAR
EXTENDS CyclicComponent IMPLEMENTS I_EtherCatMasterDiagnostic, I_Initializable, I_TaskResult, I_Simulatable
VAR
	EcMaster	AT %I*	: ST_EtherCatMasterInfo;
	FrmXWcState AT %I*	: ARRAY[0..(FRAMES - 1)] OF WORD;
	ConfiguredSlaveInfo : ARRAY[0..MAX_EC_SLAVES] OF ST_EcSlaveConfigData;
	SlavesState			: ARRAY[0..MAX_EC_SLAVES] OF ST_EcSlaveState;
	SlaveTopologyInfo	: ARRAY[0..MAX_EC_SLAVES] OF ST_TopologyDataEx;
	SyncUnit			: ARRAY[0..(SYNC_UNITS - 1)] OF SyncUnitTask('Sync Unit', THIS^, ConfiguredSlaveInfo, SlaveTopologyInfo);
	IoDevice			: ARRAY[0..MAX_EC_SLAVES] OF EtherCatIoDevice('Io Device');
	EventProvider		: I_EtherCatDiagnosticEventProvider;
END_VAR

VAR
	SlaveSequence									 : UDINT;
	RunSlaveDiag, LastFramesWcStatesOk				 : BOOL;
	LastChangeCount, LastSlaveCount, LastMasterState : UINT;
	EcStartupCycles									 : UINT;
	GetConfiguredSlaves								 : FB_EcGetConfSlaves;
	GetMasterFrameCount								 : FB_EcMasterFrameCount;
	GetAllSlaveStates								 : FB_EcGetAllSlaveStates;
	GetSlaveTopologyInfo							 : FB_EcGetSlaveTopologyInfo;
END_VAR

VAR
	{attribute 'hide'}
	_Initialized : BOOL;
	{attribute 'hide'}
	_Error : BOOL;
	{attribute 'hide'}
	_Busy : BOOL;
	{attribute 'hide'}
	_ErrorId : UDINT;
	{attribute 'hide'}
	_Simulated : BOOL;
	{attribute 'hide'}
	Config : ST_EcSlaveConfigData;
	{attribute 'hide'}
	State : ST_EcSlaveState;
	{attribute 'hide'}
	NullIoDevice : EtherCatIoDevice('NullIoDevice') := (Configuration := Config, State := State);
	{attribute 'hide'}
	_LocalAmsNetId : T_AmsNetId;
	{attribute 'hide'}
	_MasterAmsNetId : T_AmsNetId;
END_VAR

METHOD PROTECTED FramesWcStatesOk : BOOL
VAR
	i : UDINT;
END_VAR
FramesWcStatesOk := TRUE;
FOR i := 0 TO (GetMasterFrameCount.nFrames - 1) DO
	IF FrmXWcState[i] <> 0 THEN
		FramesWcStatesOk := FALSE;
		EXIT;
	END_IF
END_FOR
END_METHOD

METHOD PROTECTED LookupMasterState : STRING
VAR_INPUT
	State : UINT;
END_VAR
IF State.0 THEN
	LookupMasterState := 'Link error';
ELSIF State.1 THEN
	LookupMasterState := 'I/O locked after link error (I/O reset required)';
ELSIF State.2 THEN
	LookupMasterState := 'Link error (redundancy adapter)';
ELSIF State.3 THEN
	LookupMasterState := 'Missing one frame (redundancy mode)';
ELSIF State.4 THEN
	LookupMasterState := 'Out of send resources (I/O reset required)';
ELSIF State.5 THEN
	LookupMasterState := 'Watchdog triggered';
ELSIF State.6 THEN
	LookupMasterState := 'Ethernet driver (miniport) NOT found';
ELSIF State.7 THEN
	LookupMasterState := 'I/O reset active';
ELSIF State.8 THEN
	LookupMasterState := 'At least one device in INIT state';
ELSIF State.9 THEN
	LookupMasterState := 'At least one device in PRE-OP state';
ELSIF State.10 THEN
	LookupMasterState := 'At least one device in SAFE-OP state';
ELSIF State.11 THEN
	LookupMasterState := 'At least one device indicates an error state';
ELSIF State.12 THEN
	LookupMasterState := 'DC not in sync';
ELSE
	LookupMasterState := 'State not found';
END_IF
END_METHOD

METHOD PROTECTED LookupSlaveState : STRING
VAR_INPUT
	Slave : UINT;
END_VAR

VAR_INST
	DiagByte	: BYTE;
	BitMaskDiag : BYTE := 16#0F;
END_VAR
(* State *)
BitMaskDiag := 16#0F;
DiagByte	:= SlavesState[Slave].deviceState AND BitMaskDiag;
CASE DiagByte OF
	EC_DEVICE_STATE_INIT:
		LookupSlaveState := 'Init';

	EC_DEVICE_STATE_PREOP:
		LookupSlaveState := 'Pre-op';

	EC_DEVICE_STATE_BOOTSTRAP:
		LookupSlaveState := 'Boot';

	EC_DEVICE_STATE_SAFEOP:
		LookupSlaveState := 'Safe-op';

	EC_DEVICE_STATE_OP:
		LookupSlaveState := 'OP';

ELSE
	LookupSlaveState := '';
END_CASE

(* Additional State Bits *)
IF SlavesState[Slave].deviceState.4 THEN // EC_DEVICE_STATE_ERROR
	LookupSlaveState := CONCAT(LookupSlaveState, ' - ');
	LookupSlaveState := CONCAT(LookupSlaveState, 'State machine error in the EtherCAT slave');
END_IF

IF SlavesState[Slave].deviceState.5 THEN // EC_DEVICE_STATE_INVALID_VPRS
	LookupSlaveState := CONCAT(LookupSlaveState, ' - ');
	LookupSlaveState := CONCAT(LookupSlaveState, 'Invalid vendor ID');
END_IF

IF SlavesState[Slave].deviceState.6 THEN // EC_DEVICE_STATE_INITCMD_ERROR
	LookupSlaveState := CONCAT(LookupSlaveState, ' - ');
	LookupSlaveState := CONCAT(LookupSlaveState, 'Error during sending of initialization commands');
END_IF

IF SlavesState[Slave].deviceState.7 THEN // EC_DEVICE_STATE_DISABLED
	LookupSlaveState := CONCAT(LookupSlaveState, ' - ');
	LookupSlaveState := CONCAT(LookupSlaveState, 'Slave is disabled');
END_IF

//_____________________________________________________________________________________________________

(* Link States *)
IF SlavesState[Slave].linkState.0 THEN // EC_LINK_STATE_NOT_PRESENT
	LookupSlaveState := CONCAT(LookupSlaveState, ' - ');
	LookupSlaveState := CONCAT(LookupSlaveState, 'No EtherCAT communication with the EtherCAT slave');
END_IF

IF SlavesState[Slave].linkState.1 THEN // EC_LINK_STATE_LINK_WITHOUT_COMM
	LookupSlaveState := CONCAT(LookupSlaveState, ' - ');
	LookupSlaveState := CONCAT(LookupSlaveState, 'Error AT port X');
END_IF

IF SlavesState[Slave].linkState.2 THEN // EC_LINK_STATE_MISSING_LINK
	LookupSlaveState := CONCAT(LookupSlaveState, ' - ');
	LookupSlaveState := CONCAT(LookupSlaveState, 'Missing link AT port X');
END_IF

IF SlavesState[Slave].linkState.3 THEN // EC_LINK_STATE_ADDITIONAL_LINK
	LookupSlaveState := CONCAT(LookupSlaveState, ' - ');
	LookupSlaveState := CONCAT(LookupSlaveState, 'Additional link AT port X');
END_IF

(* Additional State Bits *)
IF SlavesState[Slave].linkState.4 THEN // EC_LINK_STATE_PORT_A
	LookupSlaveState := CONCAT(LookupSlaveState, ' - ');
	LookupSlaveState := CONCAT(LookupSlaveState, 'Port 0');
END_IF

IF SlavesState[Slave].linkState.5 THEN // EC_LINK_STATE_PORT_B
	LookupSlaveState := CONCAT(LookupSlaveState, ' - ');
	LookupSlaveState := CONCAT(LookupSlaveState, 'Port 1');
END_IF

IF SlavesState[Slave].linkState.6 THEN // EC_LINK_STATE_PORT_C
	LookupSlaveState := CONCAT(LookupSlaveState, ' - ');
	LookupSlaveState := CONCAT(LookupSlaveState, 'Port 2');
END_IF

IF SlavesState[Slave].linkState.7 THEN // EC_LINK_STATE_PORT_D
	LookupSlaveState := CONCAT(LookupSlaveState, ' - ');
	LookupSlaveState := CONCAT(LookupSlaveState, 'Port 3');
END_IF
END_METHOD

METHOD PROTECTED MasterState : BOOL
VAR_INPUT
END_VAR
IF (LastMasterState <> EcMaster.DevState) AND (EcMaster.DevState <> 0) AND (EcMaster.SlaveCount < EcMaster.CfgSlaveCount) THEN
	IF EcMaster.DevState <> 0 THEN
		IF EventProvider <> 0 THEN
			EventProvider.RaiseEtherCatDiagnosticEvent(E_EtherCatMaster.MasterError, LookupMasterState(EcMaster.DevState));
		END_IF

		_Error	 := TRUE;
		_ErrorId := EcMaster.DevState;
	END_IF
END_IF
END_METHOD

METHOD PROTECTED SlaveState : BOOL
VAR_INST
	DiagByte	 : BYTE;
	BitMaskDiag	 : BYTE := 16#0F;
	FaultedSlave : UINT;
	i, j		 : UINT;
END_VAR
CASE SlaveSequence OF
	(* Wait for start *)
	0:
		GetAllSlaveStates.bExecute	  := FALSE;
		GetSlaveTopologyInfo.bExecute := FALSE;
		IF RunSlaveDiag THEN
			RunSlaveDiag := FALSE;
			NextStep(SlaveSequence);
		END_IF

	(* Update Topology*)
	10:
		GetSlaveTopologyInfo.bExecute := TRUE;
		IF GetSlaveTopologyInfo.bBusy THEN
			NextMinorStep(SlaveSequence);
		END_IF

	11:
		IF NOT GetSlaveTopologyInfo.bBusy AND NOT GetSlaveTopologyInfo.bError THEN
			NextStep(SlaveSequence);
		END_IF

		IF GetSlaveTopologyInfo.bError THEN
			SlaveSequence := 999;
		END_IF

	(* Read Slave States *)
	20:
		GetAllSlaveStates.bExecute := TRUE;
		IF GetAllSlaveStates.bBusy THEN
			NextMinorStep(SlaveSequence);
		END_IF

	21:
		IF NOT GetAllSlaveStates.bBusy AND NOT GetAllSlaveStates.bError THEN
			NextStep(SlaveSequence);
		END_IF

		IF GetAllSlaveStates.bError THEN
			SlaveSequence := 999;
		END_IF

	(* Evaluate Slave Error *)
	30:
		FOR FaultedSlave := 0 TO (EcMaster.CfgSlaveCount - 1) DO
			BitMaskDiag := 16#0F;
			DiagByte	:= SlavesState[FaultedSlave].deviceState AND BitMaskDiag;
			IF DiagByte <> EC_DEVICE_STATE_OP AND SlaveTopologyInfo[FaultedSlave].nStatusBits.4 = FALSE THEN // No error if hotconnect
				IF SlavesState[FaultedSlave].deviceState.7 THEN												 // Slave is Disabled - warning only
					IF EventProvider <> 0 THEN
						EventProvider.RaiseEtherCatDiagnosticEvent(E_EtherCatMaster.SlaveDisabled, ConfiguredSlaveInfo[FaultedSlave].sName);
					END_IF
				ELSE
					IF EventProvider <> 0 THEN
						EventProvider.RaiseEtherCatDiagnosticEvent(E_EtherCatMaster.SlaveError, ConfiguredSlaveInfo[FaultedSlave].sName, LookupSlaveState(FaultedSlave));
					END_IF

					_Error	 := TRUE;
					_ErrorId := FaultedSlave;
					EXIT;
				END_IF
			END_IF

			BitMaskDiag := 16#0F;
			DiagByte	:= SlavesState[FaultedSlave].linkState AND BitMaskDiag;
			IF DiagByte <> EC_LINK_STATE_OK AND SlaveTopologyInfo[FaultedSlave].nStatusBits.4 = FALSE THEN // Next slave is in hotconnect group, no error
				IF EventProvider <> 0 THEN
					EventProvider.RaiseEtherCatDiagnosticEvent(E_EtherCatMaster.SlaveError, ConfiguredSlaveInfo[FaultedSlave].sName, LookupSlaveState(FaultedSlave));
				END_IF

				_Error	 := TRUE;
				_ErrorId := FaultedSlave;
				EXIT;
			END_IF
		END_FOR

		NextStep(SlaveSequence);

	(* Build Slaves *)
	40:
		FOR i := 0 TO (EcMaster.CfgSlaveCount - 1) DO
			FOR j := 0 TO (SYNC_UNITS - 1) DO
				IF SyncUnit[j].IsTerminalPartOfSyncUnit(ConfiguredSlaveInfo[i].nAddr) THEN
					IoDevice[i].SyncUnit := SyncUnit[j];
				END_IF
			END_FOR
		END_FOR

		SlaveSequence := 0;

	(* Sequence Error *)
	999:
		_ErrorId	  := 999;
		SlaveSequence := 0;
END_CASE
END_METHOD

{attribute 'monitoring' := 'call'}
PROPERTY ConfiguredSlaveCount : UINT
GET
ConfiguredSlaveCount := EcMaster.CfgSlaveCount;
END_GET
END_PROPERTY

METHOD GetIoDeviceByAddr : I_EcIoDevice
VAR_INPUT
	Addr : WORD;
END_VAR

VAR
	i : UINT;
END_VAR
IF NOT Initialized THEN
	GetIoDeviceByAddr := NullIoDevice;
	RETURN;
END_IF

FOR i := 0 TO (EcMaster.CfgSlaveCount - 1) DO
	IF IoDevice[i].Configuration.nAddr = Addr THEN
		GetIoDeviceByAddr := IoDevice[i];
		RETURN;
	END_IF
END_FOR

GetIoDeviceByAddr := NullIoDevice;
END_METHOD

METHOD GetIoDeviceByName : I_EcIoDevice
VAR_INPUT
	Name : STRING(31);
END_VAR

VAR
	i : UINT;
END_VAR
IF NOT Initialized THEN
	GetIoDeviceByName := NullIoDevice;
	RETURN;
END_IF

FOR i := 0 TO (EcMaster.CfgSlaveCount - 1) DO
	IF IoDevice[i].Name = Name THEN
		GetIoDeviceByName := IoDevice[i];
		RETURN;
	END_IF
END_FOR

GetIoDeviceByName := NullIoDevice;
END_METHOD

{attribute 'monitoring' := 'call'}
PROPERTY LocalAmsNetId : T_AmsNetId
GET
LocalAmsNetId := _LocalAmsNetId;
END_GET
END_PROPERTY

{attribute 'monitoring' := 'call'}
PROPERTY MasterAmsNetId : T_AmsNetId
GET
MasterAmsNetId := _MasterAmsNetId;
END_GET
END_PROPERTY

METHOD RegisterEventProvider
VAR_INPUT
	EventProvider : I_EtherCatDiagnosticEventProvider;
END_VAR
THIS^.EventProvider := EventProvider;
END_METHOD

{attribute 'monitoring' := 'call'}
PROPERTY SlaveCount : UINT
GET
SlaveCount := EcMaster.SlaveCount;
END_GET
END_PROPERTY

METHOD Initialize
VAR_INST
	InitSequenceState : UDINT;
	GetLocalAmsNetId  : FB_GetLocalAmsNetId;
	StartCycles		  : UINT;
END_VAR

VAR
	i : UDINT;
END_VAR
IF NOT _Error AND NOT (F_GetMappingStatus(ADR(EcMaster.AmsNetID), SIZEOF(EcMaster.AmsNetID)) <> EplcMappingStatus.MS_Unmapped) AND NOT Simulated THEN
	_Error := TRUE;
	Trace.LogMessage(Name, 'Init Failed - AmsNetID mapped to Master!');
END_IF

IF NOT _Error AND NOT (F_GetMappingStatus(ADR(EcMaster.DevID), SIZEOF(EcMaster.DevID)) <> EplcMappingStatus.MS_Unmapped) AND NOT Simulated THEN
	_Error := TRUE;
	Trace.LogMessage(Name, 'Init Failed - DevID mapped to Master!');
END_IF

IF NOT _Error AND NOT (F_GetMappingStatus(ADR(EcMaster.DevState), SIZEOF(EcMaster.DevState)) <> EplcMappingStatus.MS_Unmapped) AND NOT Simulated THEN
	_Error := TRUE;
	Trace.LogMessage(Name, 'Init Failed - DevState mapped to Master!');
END_IF

IF NOT _Error AND NOT (F_GetMappingStatus(ADR(EcMaster.ChangeCount), SIZEOF(EcMaster.ChangeCount)) <> EplcMappingStatus.MS_Unmapped) AND NOT Simulated THEN
	_Error := TRUE;
	Trace.LogMessage(Name, 'Init Failed - ChangeCount mapped to Master!');
END_IF

IF NOT _Error AND NOT (F_GetMappingStatus(ADR(EcMaster.SlaveCount), SIZEOF(EcMaster.SlaveCount)) <> EplcMappingStatus.MS_Unmapped) AND NOT Simulated THEN
	_Error := TRUE;
	Trace.LogMessage(Name, 'Init Failed - CfgSlaveCount mapped to Master!');
END_IF

IF NOT _Error AND NOT (F_GetMappingStatus(ADR(EcMaster.CfgSlaveCount), SIZEOF(EcMaster.CfgSlaveCount)) <> EplcMappingStatus.MS_Unmapped) AND NOT Simulated THEN
	_Error := TRUE;
	Trace.LogMessage(Name, 'Init Failed - CfgSlaveCount mapped to Master!');
END_IF

IF _Error THEN
	RETURN;
END_IF

IF Simulated THEN
	FOR i := 0 TO (SYNC_UNITS - 1) DO
		SyncUnit[i].EventProvider := EventProvider;
		SyncUnit[i].Simulated	  := Simulated;
		SyncUnit[i].Initialize();
		IF NOT SyncUnit[i].Initialized THEN
			RETURN;
		END_IF
	END_FOR

	_Initialized := TRUE;
	RETURN;
END_IF

GetLocalAmsNetId(tTimeOut := T#1S);
_MasterAmsNetId := F_CreateAmsNetId(EcMaster.AmsNetID);
GetMasterFrameCount(sNetId := _MasterAmsNetId, tTimeout := T#1S);
GetConfiguredSlaves(sNetId				:= _MasterAmsNetId,
					pArrEcConfSlaveInfo := ADR(ConfiguredSlaveInfo),
					cbBufLen			:= SIZEOF(ConfiguredSlaveInfo),
					tTimeout			:= T#1S);

CASE InitSequenceState OF
	0:
		GetLocalAmsNetId.bExecute := TRUE;
		IF GetLocalAmsNetId.bBusy THEN
			NextMinorStep(InitSequenceState);
		END_IF

	1:
		IF NOT GetLocalAmsNetId.bBusy AND NOT GetLocalAmsNetId.bError THEN
			_LocalAmsNetId := GetLocalAmsNetId.AddrString;
			NextStep(InitSequenceState);
		END_IF

		IF GetLocalAmsNetId.bError THEN
			_ErrorID := GetLocalAmsNetId.nErrId;
			_Error	 := TRUE;
			Trace.LogMessage(Name, 'Init Failed - GetLocalAmsNetId!');
			InitSequenceState := 999;
		END_IF

	10:
		GetConfiguredSlaves.bExecute := TRUE;
		IF GetConfiguredSlaves.bBusy THEN
			NextMinorStep(InitSequenceState);
		END_IF

	11:
		IF NOT GetConfiguredSlaves.bBusy AND NOT GetConfiguredSlaves.bError THEN
			NextStep(InitSequenceState);
		END_IF

		IF GetConfiguredSlaves.bError THEN
			_ErrorId := GetConfiguredSlaves.nErrorId;
			_Error	 := TRUE;
			Trace.LogMessage(Name, 'Init Failed - Configured EtherCat Slaves could not be read - check linking of EtherCat Master FB!');
			InitSequenceState := 999;
		END_IF

	20: // Get Master Frame Count
		GetMasterFrameCount.bExecute := TRUE;
		IF GetMasterFrameCount.bBusy THEN
			NextMinorStep(InitSequenceState);
		END_IF

	21:
		IF NOT GetMasterFrameCount.bBusy AND NOT GetMasterFrameCount.bError THEN
			// Check Frame Count
			IF GetMasterFrameCount.nFrames > FRAMES THEN
				_Error := TRUE;
				Trace.LogMessage(Name, 'Increase of Frame diagnostic array (FRAMES_MAX) and link to FrmXWcState!');
				RETURN;
			END_IF

			// Check Frame Linking
			FOR i := 0 TO (GetMasterFrameCount.nFrames - 1) DO
				IF NOT (F_GetMappingStatus(ADR(FrmXWcState[i]), SIZEOF(FrmXWcState[i])) <> EplcMappingStatus.MS_Unmapped) THEN
					_Error := TRUE;
					Trace.LogMessage(Name, 'Init Failed - FrmXWcState[x] not mapped to Master!');
					RETURN;
				END_IF
			END_FOR

			NextStep(InitSequenceState);
		END_IF

		IF GetMasterFrameCount.bError THEN
			_ErrorId := GetMasterFrameCount.nErrId;
			_Error	 := TRUE;
			Trace.LogMessage(Name, 'Init Failed - Configured EtherCat Frames could not be read!');
			InitSequenceState := 999;
		END_IF

	30:
		FOR i := 0 TO (SYNC_UNITS - 1) DO
			SyncUnit[i].EventProvider := EventProvider;
			SyncUnit[i].Initialize();
			IF NOT SyncUnit[i].Initialized THEN
				RETURN;
			END_IF
		END_FOR

		NextStep(InitSequenceState);

	40:
		StartCycles := StartCycles + 1;
		IF StartCycles = EcStartupCycles THEN
			FOR i := 0 TO (EcMaster.CfgSlaveCount - 1) DO
				IoDevice[i].AmsNetId	  := EcMaster.AmsNetID;
				IoDevice[i].Name		  := ConfiguredSlaveInfo[i].sName;
				IoDevice[i].State		  REF= SlavesState[i];
				IoDevice[i].Configuration REF= ConfiguredSlaveInfo[i];
			END_FOR

			_Initialized := TRUE;
		END_IF

	999: // Fail - Look at trace message in ADS log
END_CASE
END_METHOD

{attribute 'monitoring' := 'call'}
PROPERTY Initialized : BOOL
GET
Initialized := _Initialized;
END_GET
SET
_Initialized := Initialized;
END_SET
END_PROPERTY

METHOD Reset
IF EventProvider <> 0 THEN
	EventProvider.Reset();
END_IF

LastMasterState := 0;
LastChangeCount := 0;
LastSlaveCount	:= 0;
_Error			:= FALSE;
_ErrorId		:= 0;
SlaveSequence	:= 0;
RunSlaveDiag	:= FALSE;
END_METHOD

{attribute 'monitoring' := 'call'}
PROPERTY Busy : BOOL
GET
Busy := _Busy;
END_GET
END_PROPERTY

{attribute 'monitoring' := 'call'}
PROPERTY Error : BOOL
GET
Error := _Error;
END_GET
END_PROPERTY

{attribute 'monitoring' := 'call'}
PROPERTY ErrorId : UDINT
GET
ErrorId := _ErrorId;
END_GET
END_PROPERTY

METHOD CyclicLogic
VAR
	i : UINT;
END_VAR
IF NOT Initialized THEN
	Initialize();
	RETURN;
END_IF

IF Simulated THEN
	_Busy	 := FALSE;
	_Error	 := FALSE;
	_ErrorId := 0;
ELSE
	IF NOT _Busy THEN
		IF (LastChangeCount <> EcMaster.ChangeCount) THEN
			RunSlaveDiag := TRUE;
		ELSIF ((EcMaster.CfgSlaveCount <> EcMaster.SlaveCount) AND (LastSlaveCount <> EcMaster.SlaveCount)) THEN
			RunSlaveDiag := TRUE;
		ELSIF FramesWcStatesOk() <> LastFramesWcStatesOk THEN
			RunSlaveDiag := TRUE;
		END_IF

		IF RunSlaveDiag THEN
			LastChangeCount		 := EcMaster.ChangeCount;
			LastSlaveCount		 := EcMaster.SlaveCount;
			LastFramesWcStatesOk := FramesWcStatesOk();
		END_IF
	END_IF

	GetSlaveTopologyInfo(sNetId	  := _MasterAmsNetId,
						 pAddrBuf := ADR(SlaveTopologyInfo),
						 cbBufLen := SIZEOF(SlaveTopologyInfo),
						 tTimeout := T#5S);

	GetAllSlaveStates(sNetId	:= _MasterAmsNetId,
					  pStateBuf := ADR(SlavesState),
					  cbBufLen	:= SIZEOF(SlavesState),
					  tTimeout	:= T#5S);

	MasterState();
	SlaveState();
	FOR i := 0 TO (SYNC_UNITS - 1) DO
		SyncUnit[i].CyclicLogic();
	END_FOR

	_Busy := SlaveSequence <> 0;
END_IF

FOR i := 0 TO (EcMaster.CfgSlaveCount - 1) DO
	IoDevice[i].CyclicLogic();
END_FOR
END_METHOD

(*FB_Init is always available implicitly and it is used primarily for initialization.
The return value is not evaluated. For a specific influence, you can also declare the
methods explicitly and provide additional code there with the standard initialization
code. You can evaluate the return value.*)
METHOD FB_Init : BOOL
VAR_INPUT
	(* TRUE: the retain variables are initialized (reset warm / reset cold)*)
	bInitRetains : BOOL;

	(* TRUE: the instance will be copied to the copy code afterward (online change)   *)
	bInCopyCode		: BOOL;
	Name			: Core.T_MaxString;
	EcStartupCycles : UINT;
END_VAR
THIS^.EcStartupCycles := EcStartupCycles;
END_METHOD

{attribute 'monitoring' := 'call'}
PROPERTY Simulated : BOOL
GET
Simulated := _Simulated;
END_GET
SET
_Simulated := Simulated;
END_SET
END_PROPERTY

END_FUNCTION_BLOCK

// Components/EtherCat/SyncUnitTask
{attribute 'no_explicit_call' := 'do not call this POU directly'}
FUNCTION_BLOCK FINAL SyncUnitTask EXTENDS CyclicComponent IMPLEMENTS I_SyncUnitTask, I_Initializable, I_TaskResult, I_Simulatable
VAR
	SyncUnitTaskInfo AT %I* : ST_EtherCatSyncUnitTaskInfo;
	_SlaveCount				: UINT;
	_IsHotConnect			: BOOL;
	EcMaster				: I_EtherCatMasterDiagnostic;
	ConfiguredSlaveInfo		: REFERENCE TO ARRAY[0..MAX_EC_SLAVES] OF ST_EcSlaveConfigData;
	SlaveTopologyInfo		: REFERENCE TO ARRAY[0..MAX_EC_SLAVES] OF ST_TopologyDataEx;
	SyncUnitSlaveAddresses	: ARRAY[0..MAX_EC_SLAVES] OF UINT;
	SyncUnitSlaveNames		: ARRAY[0..MAX_EC_SLAVES] OF STRING(31);
END_VAR

VAR
	{attribute 'hide'}
	_Initialized : BOOL;
	{attribute 'hide'}
	_Error : BOOL;
	{attribute 'hide'}
	_Busy : BOOL;
	{attribute 'hide'}
	_ErrorId : UDINT;
	{attribute 'hide'}
	_Simulated : BOOL;
END_VAR

VAR
	SyncUnitState			  : UDINT := READ_SLAVES;
	i						  : UINT;
	j						  : UINT;
	_EventProvider			  : I_EtherCatDiagnosticEventProvider;
	EcGetAllSyncUnitSlaveAddr : FB_EcGetAllSyncUnitSlaveAddr;
END_VAR

VAR CONSTANT
	ERROR_READ_SLAVE_NAMES	   : UDINT := 1;
	ERROR_REGISTER_SYNC_UNIT   : UDINT := 2;
	ERROR_VALID_DATA_SYNC_UNIT : UDINT := 3;
	STRING_LEN				   : INT   := 80;
	SYNC_UNIT_ALARM_MAX		   : UINT  := 3;

	//
	READ_SLAVES			  : UDINT := 0;
	READ_SLAVES_DONE	  : UDINT := 1;
	SYNC_UNIT_OK		  : UDINT := 2;
	POPULATE_SLAVE_NAMES  : UDINT := 3;
	WORKING_COUNTER_ERROR : UDINT := 4;
	READ_ERROR			  : UDINT := 5;
END_VAR

METHOD Initialize
VAR_INPUT
END_VAR
IF NOT _Error AND NOT (F_GetMappingStatus(ADR(SyncUnitTaskInfo.ObjectId), SIZEOF(SyncUnitTaskInfo.ObjectId)) <> EplcMappingStatus.MS_Unmapped) AND NOT Simulated THEN
	_Error := TRUE;
	Trace.LogMessage(Name, 'Init Failed - SyncUnitTaskInfo.ObjectId mapped to SyncUnit Diagnostic!');
END_IF

IF NOT _Error AND NOT (F_GetMappingStatus(ADR(SyncUnitTaskInfo.SlaveCount), SIZEOF(SyncUnitTaskInfo.SlaveCount)) <> EplcMappingStatus.MS_Unmapped) AND NOT Simulated THEN
	_Error := TRUE;
	Trace.LogMessage(Name, 'Init Failed - SyncUnitTaskInfo.SlaveCount mapped to SyncUnit Diagnostic!');
END_IF

IF NOT _Error AND NOT (F_GetMappingStatus(ADR(SyncUnitTaskInfo.State), SIZEOF(SyncUnitTaskInfo.State)) <> EplcMappingStatus.MS_Unmapped) AND NOT Simulated THEN
	_Error := TRUE;
	Trace.LogMessage(Name, 'Init Failed - SyncUnitTaskInfo.State mapped to SyncUnit Diagnostic!');
END_IF

IF NOT _Error AND NOT (F_GetMappingStatus(ADR(SyncUnitTaskInfo.WcState), SIZEOF(SyncUnitTaskInfo.WcState)) <> EplcMappingStatus.MS_Unmapped) AND NOT Simulated THEN
	_Error := TRUE;
	Trace.LogMessage(Name, 'Init Failed - SyncUnitTaskInfo.WcState mapped to SyncUnit Diagnostic!');
END_IF

IF _Error THEN
	RETURN;
END_IF

IF Simulated THEN
	_Initialized := TRUE;
	RETURN;
END_IF

F_EcGetSyncUnitName(SyncUnitTaskInfo.ObjectId, sSyncUnitName => _Name);
_Initialized := TRUE;
END_METHOD

{attribute 'monitoring' := 'call'}
PROPERTY Initialized : BOOL
GET
Initialized := _Initialized;
END_GET
SET
_Initialized := Initialized;
END_SET
END_PROPERTY

{attribute 'monitoring' := 'call'}
PROPERTY IoDataValid : BOOL
GET
IoDataValid := NOT SyncUnitTaskInfo.WcState;
END_GET
END_PROPERTY

{attribute 'monitoring' := 'call'}
PROPERTY IsHotConnect : BOOL
GET
IsHotConnect := _IsHotConnect;
END_GET
END_PROPERTY

METHOD IsTerminalPartOfSyncUnit : BOOL
VAR_INPUT
	Addr : UINT;
END_VAR
FOR i := 0 TO (_SlaveCount - 1) DO
	IF SyncUnitSlaveAddresses[i] = Addr THEN
		IsTerminalPartOfSyncUnit := TRUE;
		EXIT;
	END_IF
END_FOR
END_METHOD

{attribute 'monitoring' := 'call'}
PROPERTY PUBLIC SlaveCount : UINT
GET
SlaveCount := _SlaveCount;
END_GET
END_PROPERTY

{attribute 'monitoring' := 'call'}
PROPERTY Busy : BOOL
GET
Busy := _Busy;
END_GET
END_PROPERTY

{attribute 'monitoring' := 'call'}
PROPERTY Error : BOOL
GET
Error := _Error;
END_GET
END_PROPERTY

{attribute 'monitoring' := 'call'}
PROPERTY ErrorId : UDINT
GET
ErrorId := _ErrorId;
END_GET
END_PROPERTY

METHOD PUBLIC CyclicLogic
VAR_INST
	TempSlaveMessage  : STRING;
	SlaveMessagePartA : STRING;
	SlaveMessagePartB : STRING;
END_VAR
IF NOT Initialized THEN
	Initialize();
	RETURN;
END_IF

IF Simulated THEN
	RETURN;
END_IF

EcGetAllSyncUnitSlaveAddr(sNetId	:= '',
						  nObjectId := SyncUnitTaskInfo.ObjectId,
						  pAddrBuf	:= ADR(SyncUnitSlaveAddresses),
						  cbBufLen	:= (SIZEOF(UINT) * MAX_EC_SLAVES),
						  tTimeout	:= T#5S,
						  nSlaves	=> _SlaveCount);

EcGetAllSyncUnitSlaveAddr.bExecute := FALSE;
CASE SyncUnitState OF
	READ_SLAVES:
		EcGetAllSyncUnitSlaveAddr.bExecute := TRUE;
		SyncUnitState					   := READ_SLAVES_DONE;

	READ_SLAVES_DONE:
		IF NOT EcGetAllSyncUnitSlaveAddr.bBusy AND NOT EcGetAllSyncUnitSlaveAddr.bError AND (_SlaveCount > 0) THEN
			SyncUnitState := POPULATE_SLAVE_NAMES;
		END_IF

		IF (EcGetAllSyncUnitSlaveAddr.bError OR (_SlaveCount = 0)) AND NOT EcGetAllSyncUnitSlaveAddr.bBusy THEN
			SyncUnitState := READ_ERROR;
		END_IF

